LIN {X 0,Y 355.021,Z 361.259,A -85,B 0,C 180,E1 -13509.112,E2 -13509.112} C_VEL
LIN {X 0,Y 354.928,Z 361.272,A -85,B 0,C 180,E1 -13512.581,E2 -13512.581} C_VEL
LIN {X 0,Y 354.896,Z 361.279,A -85,B 0,C 180,E1 -13516.096,E2 -13516.096} C_VEL
LIN {X 0,Y 354.913,Z 361.273,A -85,B 0,C 180,E1 -13518.472,E2 -13518.472} C_VEL
LIN {X 0,Y 354.841,Z 361.284,A -85,B 0,C 180,E1 -13522.106,E2 -13522.106} C_VEL
LIN {X 0,Y 354.905,Z 361.279,A -85,B 0,C 180,E1 -13525.827,E2 -13525.827} C_VEL
LIN {X 0,Y 354.852,Z 361.286,A -85,B 0,C 180,E1 -13529.679,E2 -13529.679} C_VEL
LIN {X 0,Y 354.812,Z 361.29,A -85,B 0,C 180,E1 -13533.702,E2 -13533.702} C_VEL
LIN {X 0,Y 354.806,Z 361.286,A -85,B 0,C 180,E1 -13536.459,E2 -13536.459} C_VEL
LIN {X 0,Y 354.83,Z 361.289,A -85,B 0,C 180,E1 -13539.423,E2 -13539.423} C_VEL
LIN {X 0,Y 354.794,Z 361.289,A -85,B 0,C 180,E1 -13542.867,E2 -13542.867} C_VEL
LIN {X 0,Y 354.786,Z 361.288,A -85,B 0,C 180,E1 -13546.106,E2 -13546.106} C_VEL
LIN {X 0,Y 354.794,Z 361.293,A -85,B 0,C 180,E1 -13549.179,E2 -13549.179} C_VEL
LIN {X 0,Y 354.813,Z 361.285,A -85,B 0,C 180,E1 -13552.402,E2 -13552.402} C_VEL
LIN {X 0,Y 354.818,Z 361.288,A -85,B 0,C 180,E1 -13554.941,E2 -13554.941} C_VEL
LIN {X 0,Y 354.799,Z 361.287,A -85,B 0,C 180,E1 -13558.405,E2 -13558.405} C_VEL
LIN {X 0,Y 354.855,Z 361.281,A -85,B 0,C 180,E1 -13561.618,E2 -13561.618} C_VEL
LIN {X 0,Y 354.905,Z 361.274,A -85,B 0,C 180,E1 -13564.172,E2 -13564.172} C_VEL
LIN {X 0,Y 354.841,Z 361.281,A -85,B 0,C 180,E1 -13567.894,E2 -13567.894} C_VEL
LIN {X 0,Y 354.928,Z 361.271,A -85,B 0,C 180,E1 -13571.891,E2 -13571.891} C_VEL
LIN {X 0,Y 354.949,Z 361.268,A -85,B 0,C 180,E1 -13575.98,E2 -13575.98} C_VEL
LIN {X 0,Y 354.974,Z 361.419,A -85,B 0,C 180,E1 -13578.978,E2 -13578.978} C_VEL
LIN {X 0,Y 358.596,Z 373.086,A -85,B 0,C 180,E1 -13579.84,E2 -13579.84} C_VEL
LIN {X 0,Y 360.664,Z 380.509,A -85,B 0,C 180,E1 -13580.491,E2 -13580.491} C_VEL
LIN {X 0,Y 359.761,Z 392.776,A -85,B 0,C 180,E1 -13581.574,E2 -13581.574} C_VEL
LIN {X 0,Y 358.877,Z 403.838,A -85,B 0,C 180,E1 -13582.827,E2 -13582.827} C_VEL
LIN {X 0,Y 358.135,Z 412.74,A -85,B 0,C 180,E1 -13584.086,E2 -13584.086} C_VEL
LIN {X 0,Y 357.355,Z 420.912,A -85,B 0,C 180,E1 -13585.487,E2 -13585.487} C_VEL
LIN {X 0,Y 356.477,Z 428.926,A -85,B 0,C 180,E1 -13587.174,E2 -13587.174} C_VEL
LIN {X 0,Y 355.809,Z 435.373,A -85,B 0,C 180,E1 -13588.867,E2 -13588.867} C_VEL
LIN {X 0,Y 355.327,Z 440.508,A -85,B 0,C 180,E1 -13590.566,E2 -13590.566} C_VEL
LIN {X 0,Y 354.88,Z 444.523,A -85,B 0,C 180,E1 -13592.269,E2 -13592.269} C_VEL
LIN {X 0,Y 354.623,Z 446.627,A -85,B 0,C 180,E1 -13593.408,E2 -13593.408} C_VEL
LIN {X 0,Y 354.558,Z 449.523,A -85,B 0,C 180,E1 -13595.687,E2 -13595.687} C_VEL
LIN {X 0,Y 354.54,Z 450.755,A -85,B 0,C 180,E1 -13597.626,E2 -13597.626} C_VEL
LIN {X 0,Y 354.539,Z 450.924,A -85,B 0,C 180,E1 -13599.124,E2 -13599.124} C_VEL
LIN {X 0,Y 354.762,Z 449.92,A -85,B 0,C 180,E1 -13601.425,E2 -13601.425} C_VEL
LIN {X 0,Y 354.949,Z 448.782,A -85,B 0,C 180,E1 -13602.579,E2 -13602.579} C_VEL
LIN {X 0,Y 355.473,Z 446.222,A -85,B 0,C 180,E1 -13604.354,E2 -13604.354} C_VEL
LIN {X 0,Y 356.044,Z 442.817,A -85,B 0,C 180,E1 -13606.042,E2 -13606.042} C_VEL
LIN {X 0,Y 356.747,Z 438.198,A -85,B 0,C 180,E1 -13607.779,E2 -13607.779} C_VEL
LIN {X 0,Y 357.852,Z 431.183,A -85,B 0,C 180,E1 -13609.802,E2 -13609.802} C_VEL
LIN {X 0,Y 359.004,Z 423.471,A -85,B 0,C 180,E1 -13611.533,E2 -13611.533} C_VEL
LIN {X 0,Y 360.247,Z 414.193,A -85,B 0,C 180,E1 -13613.19,E2 -13613.19} C_VEL
LIN {X 0,Y 361.309,Z 404.665,A -85,B 0,C 180,E1 -13614.567,E2 -13614.567} C_VEL
LIN {X 0,Y 362.351,Z 394.731,A -85,B 0,C 180,E1 -13615.719,E2 -13615.719} C_VEL
LIN {X 0,Y 363.291,Z 385.09,A -85,B 0,C 180,E1 -13616.62,E2 -13616.62} C_VEL
LIN {X 0,Y 359.553,Z 373.52,A -85,B 0,C 180,E1 -13617.813,E2 -13617.813} C_VEL
LIN {X 0,Y 354.995,Z 361.878,A -85,B 0,C 180,E1 -13618.848,E2 -13618.848} C_VEL
LIN {X 0,Y 354.862,Z 361.284,A -85,B 0,C 180,E1 -13618.947,E2 -13618.947} C_VEL
LIN {X 0,Y 354.788,Z 361.299,A -85,B 0,C 180,E1 -13622.332,E2 -13622.332} C_VEL
LIN {X 0,Y 354.822,Z 361.291,A -85,B 0,C 180,E1 -13625.698,E2 -13625.698} C_VEL
LIN {X 0,Y 354.824,Z 361.288,A -85,B 0,C 180,E1 -13629.423,E2 -13629.423} C_VEL
LIN {X 0,Y 354.779,Z 361.293,A -85,B 0,C 180,E1 -13631.346,E2 -13631.346} C_VEL
LIN {X 0,Y 354.081,Z 361.38,A -85,B 0,C 180,E1 -13632.293,E2 -13632.293} C_VEL
LIN {X 0,Y 351.182,Z 361.741,A -85,B 0,C 180,E1 -13633.831,E2 -13633.831} C_VEL
LIN {X 0,Y 348.77,Z 362.043,A -85,B 0,C 180,E1 -13635.076,E2 -13635.076} C_VEL
LIN {X 0,Y 347.779,Z 362.167,A -85,B 0,C 180,E1 -13636.04,E2 -13636.04} C_VEL
LIN {X 0,Y 347.721,Z 362.17,A -85,B 0,C 180,E1 -13636.367,E2 -13636.367} C_VEL
LIN {X 0,Y 347.754,Z 362.168,A -85,B 0,C 180,E1 -13639.705,E2 -13639.705} C_VEL
LIN {X 0,Y 347.765,Z 362.167,A -85,B 0,C 180,E1 -13642.679,E2 -13642.679} C_VEL
LIN {X 0,Y 347.746,Z 362.17,A -85,B 0,C 180,E1 -13645.955,E2 -13645.955} C_VEL
LIN {X 0,Y 347.768,Z 362.134,A -85,B 0,C 180,E1 -13649.653,E2 -13649.653} C_VEL
LIN {X 0,Y 347.85,Z 362.149,A -85,B 0,C 180,E1 -13652.744,E2 -13652.744} C_VEL
LIN {X 0,Y 347.785,Z 362.157,A -85,B 0,C 180,E1 -13656.161,E2 -13656.161} C_VEL
LIN {X 0,Y 347.814,Z 362.16,A -85,B 0,C 180,E1 -13659.909,E2 -13659.909} C_VEL
LIN {X 0,Y 347.863,Z 362.145,A -85,B 0,C 180,E1 -13662.359,E2 -13662.359} C_VEL
LIN {X 0,Y 347.894,Z 362.151,A -85,B 0,C 180,E1 -13665.97,E2 -13665.97} C_VEL
LIN {X 0,Y 347.93,Z 362.144,A -85,B 0,C 180,E1 -13669.525,E2 -13669.525} C_VEL
LIN {X 0,Y 348.071,Z 362.129,A -85,B 0,C 180,E1 -13671.874,E2 -13671.874} C_VEL
LIN {X 0,Y 348.065,Z 362.118,A -85,B 0,C 180,E1 -13674.205,E2 -13674.205} C_VEL
LIN {X 0,Y 348.205,Z 362.112,A -85,B 0,C 180,E1 -13677.686,E2 -13677.686} C_VEL
LIN {X 0,Y 348.365,Z 362.082,A -85,B 0,C 180,E1 -13680,E2 -13680} C_VEL
LIN {X 0,Y 348.205,Z 362.113,A -85,B 0,C 180,E1 -13682.313,E2 -13682.313} C_VEL
LIN {X 0,Y 348.102,Z 362.124,A -85,B 0,C 180,E1 -13686.957,E2 -13686.957} C_VEL
LIN {X 0,Y 347.963,Z 362.136,A -85,B 0,C 180,E1 -13689.298,E2 -13689.298} C_VEL
LIN {X 0,Y 347.886,Z 362.15,A -85,B 0,C 180,E1 -13692.839,E2 -13692.839} C_VEL
LIN {X 0,Y 347.835,Z 362.158,A -85,B 0,C 180,E1 -13696.431,E2 -13696.431} C_VEL
LIN {X 0,Y 347.851,Z 362.156,A -85,B 0,C 180,E1 -13698.86,E2 -13698.86} C_VEL
LIN {X 0,Y 347.77,Z 362.168,A -85,B 0,C 180,E1 -13702.579,E2 -13702.579} C_VEL
LIN {X 0,Y 347.808,Z 362.165,A -85,B 0,C 180,E1 -13705.109,E2 -13705.109} C_VEL
LIN {X 0,Y 347.808,Z 362.165,A -85,B 0,C 180,E1 -13707.694,E2 -13707.694} C_VEL
LIN {X 0,Y 347.76,Z 362.171,A -85,B 0,C 180,E1 -13710.347,E2 -13710.347} C_VEL
LIN {X 0,Y 347.741,Z 362.171,A -85,B 0,C 180,E1 -13714.464,E2 -13714.464} C_VEL
LIN {X 0,Y 347.776,Z 362.156,A -85,B 0,C 180,E1 -13717.99,E2 -13717.99} C_VEL
LIN {X 0,Y 347.78,Z 362.155,A -85,B 0,C 180,E1 -13721.826,E2 -13721.826} C_VEL
LIN {X 0,Y 347.797,Z 362.164,A -85,B 0,C 180,E1 -13722.213,E2 -13722.213} C_VEL
LIN {X 0,Y 349.191,Z 369.057,A -85,B 0,C 180,E1 -13725.701,E2 -13725.701} C_VEL
LIN {X 0,Y 350.381,Z 375.055,A -85,B 0,C 180,E1 -13728.555,E2 -13728.555} C_VEL
LIN {X 0,Y 351.655,Z 382.173,A -85,B 0,C 180,E1 -13731.718,E2 -13731.718} C_VEL
LIN {X 0,Y 351.741,Z 385.397,A -85,B 0,C 180,E1 -13733.056,E2 -13733.056} C_VEL
LIN {X 0,Y 350.275,Z 396.112,A -85,B 0,C 180,E1 -13737.199,E2 -13737.199} C_VEL
LIN {X 0,Y 349.041,Z 406.501,A -85,B 0,C 180,E1 -13741.104,E2 -13741.104} C_VEL
LIN {X 0,Y 348.092,Z 416.889,A -85,B 0,C 180,E1 -13744.914,E2 -13744.914} C_VEL
LIN {X 0,Y 347.423,Z 425.713,A -85,B 0,C 180,E1 -13748.105,E2 -13748.105} C_VEL
LIN {X 0,Y 350.097,Z 440.51,A -85,B 0,C 180,E1 -13748.818,E2 -13748.818} C_VEL
LIN {X 0,Y 351.654,Z 453.114,A -85,B 0,C 180,E1 -13749.614,E2 -13749.614} C_VEL
LIN {X 0,Y 352.322,Z 464.451,A -85,B 0,C 180,E1 -13750.489,E2 -13750.489} C_VEL
LIN {X 0,Y 352.267,Z 477.128,A -85,B 0,C 180,E1 -13751.687,E2 -13751.687} C_VEL
LIN {X 0,Y 351.127,Z 487.251,A -85,B 0,C 180,E1 -13752.83,E2 -13752.83} C_VEL
LIN {X 0,Y 349.685,Z 497.503,A -85,B 0,C 180,E1 -13754.258,E2 -13754.258} C_VEL
LIN {X 0,Y 348.829,Z 505.758,A -85,B 0,C 180,E1 -13755.677,E2 -13755.677} C_VEL
LIN {X 0,Y 347.695,Z 514.218,A -85,B 0,C 180,E1 -13757.451,E2 -13757.451} C_VEL
LIN {X 0,Y 346.983,Z 520.939,A -85,B 0,C 180,E1 -13759.202,E2 -13759.202} C_VEL
LIN {X 0,Y 346.652,Z 527.13,A -85,B 0,C 180,E1 -13761.255,E2 -13761.255} C_VEL
LIN {X 0,Y 346.637,Z 532.039,A -85,B 0,C 180,E1 -13763.447,E2 -13763.447} C_VEL
LIN {X 0,Y 346.765,Z 535.029,A -85,B 0,C 180,E1 -13765.351,E2 -13765.351} C_VEL
LIN {X 0,Y 346.931,Z 536.325,A -85,B 0,C 180,E1 -13766.517,E2 -13766.517} C_VEL
LIN {X 0,Y 346.964,Z 537.152,A -85,B 0,C 180,E1 -13767.679,E2 -13767.679} C_VEL
LIN {X 0,Y 347.059,Z 537.594,A -85,B 0,C 180,E1 -13770.001,E2 -13770.001} C_VEL
LIN {X 0,Y 347.019,Z 537.206,A -85,B 0,C 180,E1 -13771.161,E2 -13771.161} C_VEL
LIN {X 0,Y 347.012,Z 536.375,A -85,B 0,C 180,E1 -13772.322,E2 -13772.322} C_VEL
LIN {X 0,Y 347.078,Z 535.124,A -85,B 0,C 180,E1 -13773.484,E2 -13773.484} C_VEL
LIN {X 0,Y 346.836,Z 532.39,A -85,B 0,C 180,E1 -13775.233,E2 -13775.233} C_VEL
LIN {X 0,Y 346.749,Z 528.611,A -85,B 0,C 180,E1 -13776.986,E2 -13776.986} C_VEL
LIN {X 0,Y 346.752,Z 523.674,A -85,B 0,C 180,E1 -13778.744,E2 -13778.744} C_VEL
LIN {X 0,Y 346.95,Z 517.446,A -85,B 0,C 180,E1 -13780.505,E2 -13780.505} C_VEL
LIN {X 0,Y 347.514,Z 509.73,A -85,B 0,C 180,E1 -13782.261,E2 -13782.261} C_VEL
LIN {X 0,Y 348.231,Z 501.871,A -85,B 0,C 180,E1 -13783.719,E2 -13783.719} C_VEL
LIN {X 0,Y 348.864,Z 494.15,A -85,B 0,C 180,E1 -13784.913,E2 -13784.913} C_VEL
LIN {X 0,Y 349.834,Z 484.267,A -85,B 0,C 180,E1 -13786.186,E2 -13786.186} C_VEL
LIN {X 0,Y 350.586,Z 474.636,A -85,B 0,C 180,E1 -13787.199,E2 -13787.199} C_VEL
LIN {X 0,Y 350.156,Z 462.196,A -85,B 0,C 180,E1 -13788.278,E2 -13788.278} C_VEL
LIN {X 0,Y 349.338,Z 449.493,A -85,B 0,C 180,E1 -13789.136,E2 -13789.136} C_VEL
LIN {X 0,Y 348.224,Z 436.683,A -85,B 0,C 180,E1 -13789.778,E2 -13789.778} C_VEL
LIN {X 0,Y 347.061,Z 426.898,A -85,B 0,C 180,E1 -13790.137,E2 -13790.137} C_VEL
LIN {X 0,Y 347.661,Z 415.33,A -85,B 0,C 180,E1 -13794.205,E2 -13794.205} C_VEL
LIN {X 0,Y 348.503,Z 403.834,A -85,B 0,C 180,E1 -13798.289,E2 -13798.289} C_VEL
LIN {X 0,Y 349.388,Z 393.64,A -85,B 0,C 180,E1 -13801.955,E2 -13801.955} C_VEL
LIN {X 0,Y 350.621,Z 382.261,A -85,B 0,C 180,E1 -13806.148,E2 -13806.148} C_VEL
LIN {X 0,Y 350.742,Z 378.306,A -85,B 0,C 180,E1 -13807.673,E2 -13807.673} C_VEL
LIN {X 0,Y 349.416,Z 370.597,A -85,B 0,C 180,E1 -13810.852,E2 -13810.852} C_VEL
LIN {X 0,Y 347.922,Z 362.984,A -85,B 0,C 180,E1 -13814.185,E2 -13814.185} C_VEL
LIN {X 0,Y 347.794,Z 362.167,A -85,B 0,C 180,E1 -13814.577,E2 -13814.577} C_VEL
LIN {X 0,Y 347.754,Z 362.165,A -85,B 0,C 180,E1 -13818.398,E2 -13818.398} C_VEL
LIN {X 0,Y 347.778,Z 362.161,A -85,B 0,C 180,E1 -13822.012,E2 -13822.012} C_VEL
LIN {X 0,Y 347.749,Z 362.165,A -85,B 0,C 180,E1 -13825.537,E2 -13825.537} C_VEL
LIN {X 0,Y 347.749,Z 362.166,A -85,B 0,C 180,E1 -13828.301,E2 -13828.301} C_VEL
LIN {X 0,Y 347.783,Z 362.164,A -85,B 0,C 180,E1 -13830.988,E2 -13830.988} C_VEL
LIN {X 0,Y 347.836,Z 362.154,A -85,B 0,C 180,E1 -13833.608,E2 -13833.608} C_VEL
LIN {X 0,Y 347.794,Z 362.16,A -85,B 0,C 180,E1 -13836.162,E2 -13836.162} C_VEL
LIN {X 0,Y 347.818,Z 362.157,A -85,B 0,C 180,E1 -13839.91,E2 -13839.91} C_VEL
LIN {X 0,Y 347.871,Z 362.153,A -85,B 0,C 180,E1 -13842.36,E2 -13842.36} C_VEL
LIN {X 0,Y 347.903,Z 362.147,A -85,B 0,C 180,E1 -13845.971,E2 -13845.971} C_VEL
LIN {X 0,Y 347.934,Z 362.142,A -85,B 0,C 180,E1 -13849.526,E2 -13849.526} C_VEL
LIN {X 0,Y 348.114,Z 362.12,A -85,B 0,C 180,E1 -13853.043,E2 -13853.043} C_VEL
LIN {X 0,Y 348.211,Z 362.108,A -85,B 0,C 180,E1 -13857.687,E2 -13857.687} C_VEL
LIN {X 0,Y 348.352,Z 362.093,A -85,B 0,C 180,E1 -13860,E2 -13860} C_VEL
LIN {X 0,Y 348.212,Z 362.112,A -85,B 0,C 180,E1 -13862.314,E2 -13862.314} C_VEL
LIN {X 0,Y 348.112,Z 362.119,A -85,B 0,C 180,E1 -13866.958,E2 -13866.958} C_VEL
LIN {X 0,Y 347.974,Z 362.137,A -85,B 0,C 180,E1 -13869.299,E2 -13869.299} C_VEL
LIN {X 0,Y 347.896,Z 362.146,A -85,B 0,C 180,E1 -13872.84,E2 -13872.84} C_VEL
LIN {X 0,Y 347.845,Z 362.154,A -85,B 0,C 180,E1 -13876.431,E2 -13876.431} C_VEL
LIN {X 0,Y 347.862,Z 362.15,A -85,B 0,C 180,E1 -13878.86,E2 -13878.86} C_VEL
LIN {X 0,Y 347.78,Z 362.161,A -85,B 0,C 180,E1 -13882.579,E2 -13882.579} C_VEL
LIN {X 0,Y 347.818,Z 362.157,A -85,B 0,C 180,E1 -13885.108,E2 -13885.108} C_VEL
LIN {X 0,Y 347.814,Z 362.163,A -85,B 0,C 180,E1 -13887.694,E2 -13887.694} C_VEL
LIN {X 0,Y 347.767,Z 362.163,A -85,B 0,C 180,E1 -13890.347,E2 -13890.347} C_VEL
LIN {X 0,Y 347.75,Z 362.164,A -85,B 0,C 180,E1 -13894.464,E2 -13894.464} C_VEL
LIN {X 0,Y 347.782,Z 362.162,A -85,B 0,C 180,E1 -13897.989,E2 -13897.989} C_VEL
LIN {X 0,Y 347.757,Z 362.166,A -85,B 0,C 180,E1 -13901.83,E2 -13901.83} C_VEL
LIN {X 0,Y 347.772,Z 362.165,A -85,B 0,C 180,E1 -13905.017,E2 -13905.017} C_VEL
LIN {X 0,Y 347.756,Z 362.164,A -85,B 0,C 180,E1 -13908.397,E2 -13908.397} C_VEL
LIN {X 0,Y 347.78,Z 362.161,A -85,B 0,C 180,E1 -13912.011,E2 -13912.011} C_VEL
LIN {X 0,Y 347.75,Z 362.167,A -85,B 0,C 180,E1 -13915.536,E2 -13915.536} C_VEL
LIN {X 0,Y 347.77,Z 362.163,A -85,B 0,C 180,E1 -13919.653,E2 -13919.653} C_VEL
LIN {X 0,Y 347.857,Z 362.155,A -85,B 0,C 180,E1 -13922.744,E2 -13922.744} C_VEL
LIN {X 0,Y 347.795,Z 362.159,A -85,B 0,C 180,E1 -13926.161,E2 -13926.161} C_VEL
LIN {X 0,Y 347.819,Z 362.156,A -85,B 0,C 180,E1 -13929.909,E2 -13929.909} C_VEL
LIN {X 0,Y 347.872,Z 362.151,A -85,B 0,C 180,E1 -13932.359,E2 -13932.359} C_VEL
LIN {X 0,Y 347.903,Z 362.146,A -85,B 0,C 180,E1 -13935.97,E2 -13935.97} C_VEL
LIN {X 0,Y 347.931,Z 362.337,A -85,B 0,C 180,E1 -13938.64,E2 -13938.64} C_VEL
LIN {X 0,Y 351.521,Z 373.703,A -85,B 0,C 180,E1 -13939.502,E2 -13939.502} C_VEL
LIN {X 0,Y 353.811,Z 381.971,A -85,B 0,C 180,E1 -13940.247,E2 -13940.247} C_VEL
LIN {X 0,Y 352.949,Z 393.281,A -85,B 0,C 180,E1 -13941.266,E2 -13941.266} C_VEL
LIN {X 0,Y 352.034,Z 404.422,A -85,B 0,C 180,E1 -13942.543,E2 -13942.543} C_VEL
LIN {X 0,Y 351.159,Z 414.255,A -85,B 0,C 180,E1 -13943.968,E2 -13943.968} C_VEL
LIN {X 0,Y 350.215,Z 423.775,A -85,B 0,C 180,E1 -13945.683,E2 -13945.683} C_VEL
LIN {X 0,Y 349.335,Z 431.411,A -85,B 0,C 180,E1 -13947.405,E2 -13947.405} C_VEL
LIN {X 0,Y 348.585,Z 438.404,A -85,B 0,C 180,E1 -13949.422,E2 -13949.422} C_VEL
LIN {X 0,Y 348.098,Z 443.08,A -85,B 0,C 180,E1 -13951.156,E2 -13951.156} C_VEL
LIN {X 0,Y 347.72,Z 446.676,A -85,B 0,C 180,E1 -13952.895,E2 -13952.895} C_VEL
LIN {X 0,Y 347.543,Z 449.272,A -85,B 0,C 180,E1 -13954.639,E2 -13954.639} C_VEL
LIN {X 0,Y 347.516,Z 450.499,A -85,B 0,C 180,E1 -13955.803,E2 -13955.803} C_VEL
LIN {X 0,Y 347.49,Z 451.631,A -85,B 0,C 180,E1 -13957.677,E2 -13957.677} C_VEL
LIN {X 0,Y 347.527,Z 451.784,A -85,B 0,C 180,E1 -13959.31,E2 -13959.31} C_VEL
LIN {X 0,Y 347.61,Z 451.448,A -85,B 0,C 180,E1 -13960.483,E2 -13960.483} C_VEL
LIN {X 0,Y 347.763,Z 450.703,A -85,B 0,C 180,E1 -13961.658,E2 -13961.658} C_VEL
LIN {X 0,Y 347.981,Z 449.527,A -85,B 0,C 180,E1 -13962.835,E2 -13962.835} C_VEL
LIN {X 0,Y 348.492,Z 447.114,A -85,B 0,C 180,E1 -13964.529,E2 -13964.529} C_VEL
LIN {X 0,Y 349.148,Z 443.435,A -85,B 0,C 180,E1 -13966.367,E2 -13966.367} C_VEL
LIN {X 0,Y 349.912,Z 438.745,A -85,B 0,C 180,E1 -13968.138,E2 -13968.138} C_VEL
LIN {X 0,Y 350.913,Z 432.759,A -85,B 0,C 180,E1 -13969.905,E2 -13969.905} C_VEL
LIN {X 0,Y 352.103,Z 425.256,A -85,B 0,C 180,E1 -13971.669,E2 -13971.669} C_VEL
LIN {X 0,Y 353.213,Z 417.516,A -85,B 0,C 180,E1 -13973.139,E2 -13973.139} C_VEL
LIN {X 0,Y 354.387,Z 407.977,A -85,B 0,C 180,E1 -13974.61,E2 -13974.61} C_VEL
LIN {X 0,Y 355.626,Z 397.404,A -85,B 0,C 180,E1 -13975.915,E2 -13975.915} C_VEL
LIN {X 0,Y 356.659,Z 386.918,A -85,B 0,C 180,E1 -13976.949,E2 -13976.949} C_VEL
LIN {X 0,Y 353.253,Z 376.293,A -85,B 0,C 180,E1 -13978.104,E2 -13978.104} C_VEL
LIN {X 0,Y 348.435,Z 364.327,A -85,B 0,C 180,E1 -13979.24,E2 -13979.24} C_VEL
LIN {X 0,Y 347.781,Z 362.17,A -85,B 0,C 180,E1 -13979.446,E2 -13979.446} C_VEL
LIN {X 0,Y 347.733,Z 362.172,A -85,B 0,C 180,E1 -13983.071,E2 -13983.071} C_VEL
LIN {X 0,Y 347.77,Z 362.168,A -85,B 0,C 180,E1 -13986.064,E2 -13986.064} C_VEL
LIN {X 0,Y 347.752,Z 362.171,A -85,B 0,C 180,E1 -13988.792,E2 -13988.792} C_VEL
LIN {X 0,Y 347.75,Z 362.167,A -85,B 0,C 180,E1 -13991.829,E2 -13991.829} C_VEL
LIN {X 0,Y 347.708,Z 362.175,A -85,B 0,C 180,E1 -13995.025,E2 -13995.025} C_VEL
LIN {X 0,Y 347.721,Z 362.17,A -85,B 0,C 180,E1 -13996.367,E2 -13996.367} C_VEL
LIN {X 0,Y 347.104,Z 362.251,A -85,B 0,C 180,E1 -13997.334,E2 -13997.334} C_VEL
LIN {X 0,Y 344.233,Z 362.61,A -85,B 0,C 180,E1 -13998.907,E2 -13998.907} C_VEL
LIN {X 0,Y 341.79,Z 362.909,A -85,B 0,C 180,E1 -14000.181,E2 -14000.181} C_VEL
LIN {X 0,Y 340.774,Z 363.039,A -85,B 0,C 180,E1 -14001.168,E2 -14001.168} C_VEL
LIN {X 0,Y 340.71,Z 363.048,A -85,B 0,C 180,E1 -14001.502,E2 -14001.502} C_VEL
LIN {X 0,Y 340.717,Z 363.045,A -85,B 0,C 180,E1 -14004.72,E2 -14004.72} C_VEL
LIN {X 0,Y 340.714,Z 363.017,A -85,B 0,C 180,E1 -14008.956,E2 -14008.956} C_VEL
LIN {X 0,Y 340.777,Z 363.028,A -85,B 0,C 180,E1 -14012.473,E2 -14012.473} C_VEL
LIN {X 0,Y 340.753,Z 363.036,A -85,B 0,C 180,E1 -14015.638,E2 -14015.638} C_VEL
LIN {X 0,Y 340.753,Z 363.041,A -85,B 0,C 180,E1 -14019.474,E2 -14019.474} C_VEL
LIN {X 0,Y 340.855,Z 363.018,A -85,B 0,C 180,E1 -14021.984,E2 -14021.984} C_VEL
LIN {X 0,Y 340.865,Z 363.026,A -85,B 0,C 180,E1 -14025.704,E2 -14025.704} C_VEL
LIN {X 0,Y 340.872,Z 363.024,A -85,B 0,C 180,E1 -14029.306,E2 -14029.306} C_VEL
LIN {X 0,Y 341.072,Z 362.997,A -85,B 0,C 180,E1 -14032.898,E2 -14032.898} C_VEL
LIN {X 0,Y 341.167,Z 362.988,A -85,B 0,C 180,E1 -14037.638,E2 -14037.638} C_VEL
LIN {X 0,Y 341.314,Z 362.96,A -85,B 0,C 180,E1 -14040,E2 -14040} C_VEL
LIN {X 0,Y 341.167,Z 362.99,A -85,B 0,C 180,E1 -14042.361,E2 -14042.361} C_VEL
LIN {X 0,Y 341.072,Z 363.001,A -85,B 0,C 180,E1 -14047.102,E2 -14047.102} C_VEL
LIN {X 0,Y 340.867,Z 363.022,A -85,B 0,C 180,E1 -14050.694,E2 -14050.694} C_VEL
LIN {X 0,Y 340.858,Z 363.021,A -85,B 0,C 180,E1 -14054.325,E2 -14054.325} C_VEL
LIN {X 0,Y 340.833,Z 363.029,A -85,B 0,C 180,E1 -14058.467,E2 -14058.467} C_VEL
LIN {X 0,Y 340.749,Z 363.042,A -85,B 0,C 180,E1 -14061.857,E2 -14061.857} C_VEL
LIN {X 0,Y 340.769,Z 363.041,A -85,B 0,C 180,E1 -14065.665,E2 -14065.665} C_VEL
LIN {X 0,Y 340.738,Z 363.045,A -85,B 0,C 180,E1 -14068.32,E2 -14068.32} C_VEL
LIN {X 0,Y 340.7,Z 363.049,A -85,B 0,C 180,E1 -14071.044,E2 -14071.044} C_VEL
LIN {X 0,Y 340.715,Z 363.044,A -85,B 0,C 180,E1 -14075.279,E2 -14075.279} C_VEL
LIN {X 0,Y 340.716,Z 363.033,A -85,B 0,C 180,E1 -14078.389,E2 -14078.389} C_VEL
LIN {X 0,Y 340.764,Z 363.119,A -85,B 0,C 180,E1 -14081.701,E2 -14081.701} C_VEL
LIN {X 0,Y 342.074,Z 369.494,A -85,B 0,C 180,E1 -14085.041,E2 -14085.041} C_VEL
LIN {X 0,Y 343.401,Z 376.226,A -85,B 0,C 180,E1 -14088.319,E2 -14088.319} C_VEL
LIN {X 0,Y 344.686,Z 383.399,A -85,B 0,C 180,E1 -14091.588,E2 -14091.588} C_VEL
LIN {X 0,Y 344.839,Z 385.866,A -85,B 0,C 180,E1 -14092.64,E2 -14092.64} C_VEL
LIN {X 0,Y 343.457,Z 395.449,A -85,B 0,C 180,E1 -14096.463,E2 -14096.463} C_VEL
LIN {X 0,Y 342.136,Z 405.829,A -85,B 0,C 180,E1 -14100.463,E2 -14100.463} C_VEL
LIN {X 0,Y 341.152,Z 416.18,A -85,B 0,C 180,E1 -14104.367,E2 -14104.367} C_VEL
LIN {X 0,Y 340.455,Z 424.893,A -85,B 0,C 180,E1 -14107.57,E2 -14107.57} C_VEL
LIN {X 0,Y 343.155,Z 439.246,A -85,B 0,C 180,E1 -14108.286,E2 -14108.286} C_VEL
LIN {X 0,Y 344.743,Z 451.758,A -85,B 0,C 180,E1 -14109.091,E2 -14109.091} C_VEL
LIN {X 0,Y 345.479,Z 463.306,A -85,B 0,C 180,E1 -14110.003,E2 -14110.003} C_VEL
LIN {X 0,Y 345.44,Z 475.363,A -85,B 0,C 180,E1 -14111.158,E2 -14111.158} C_VEL
LIN {X 0,Y 344.857,Z 483.284,A -85,B 0,C 180,E1 -14112.048,E2 -14112.048} C_VEL
LIN {X 0,Y 343.333,Z 493.137,A -85,B 0,C 180,E1 -14113.348,E2 -14113.348} C_VEL
LIN {X 0,Y 342.02,Z 503.004,A -85,B 0,C 180,E1 -14114.968,E2 -14114.968} C_VEL
LIN {X 0,Y 341.233,Z 509.666,A -85,B 0,C 180,E1 -14116.3,E2 -14116.3} C_VEL
LIN {X 0,Y 340.326,Z 517.087,A -85,B 0,C 180,E1 -14118.083,E2 -14118.083} C_VEL
LIN {X 0,Y 339.753,Z 523.084,A -85,B 0,C 180,E1 -14119.874,E2 -14119.874} C_VEL
LIN {X 0,Y 339.543,Z 527.863,A -85,B 0,C 180,E1 -14121.67,E2 -14121.67} C_VEL
LIN {X 0,Y 339.561,Z 531.518,A -85,B 0,C 180,E1 -14123.449,E2 -14123.449} C_VEL
LIN {X 0,Y 339.682,Z 534.216,A -85,B 0,C 180,E1 -14125.254,E2 -14125.254} C_VEL
LIN {X 0,Y 339.857,Z 535.491,A -85,B 0,C 180,E1 -14126.444,E2 -14126.444} C_VEL
LIN {X 0,Y 339.915,Z 536.3,A -85,B 0,C 180,E1 -14127.631,E2 -14127.631} C_VEL
LIN {X 0,Y 340.013,Z 536.714,A -85,B 0,C 180,E1 -14130.001,E2 -14130.001} C_VEL
LIN {X 0,Y 339.971,Z 536.306,A -85,B 0,C 180,E1 -14131.185,E2 -14131.185} C_VEL
LIN {X 0,Y 339.966,Z 535.449,A -85,B 0,C 180,E1 -14132.37,E2 -14132.37} C_VEL
LIN {X 0,Y 340.033,Z 534.182,A -85,B 0,C 180,E1 -14133.556,E2 -14133.556} C_VEL
LIN {X 0,Y 339.761,Z 531.411,A -85,B 0,C 180,E1 -14135.342,E2 -14135.342} C_VEL
LIN {X 0,Y 339.693,Z 527.597,A -85,B 0,C 180,E1 -14137.132,E2 -14137.132} C_VEL
LIN {X 0,Y 339.684,Z 522.618,A -85,B 0,C 180,E1 -14138.928,E2 -14138.928} C_VEL
LIN {X 0,Y 339.917,Z 516.348,A -85,B 0,C 180,E1 -14140.725,E2 -14140.725} C_VEL
LIN {X 0,Y 340.506,Z 508.583,A -85,B 0,C 180,E1 -14142.517,E2 -14142.517} C_VEL
LIN {X 0,Y 341.22,Z 500.655,A -85,B 0,C 180,E1 -14144.006,E2 -14144.006} C_VEL
LIN {X 0,Y 342.196,Z 490.991,A -85,B 0,C 180,E1 -14145.486,E2 -14145.486} C_VEL
LIN {X 0,Y 343.195,Z 480.271,A -85,B 0,C 180,E1 -14146.814,E2 -14146.814} C_VEL
LIN {X 0,Y 343.567,Z 474.633,A -85,B 0,C 180,E1 -14147.409,E2 -14147.409} C_VEL
LIN {X 0,Y 343.206,Z 462.733,A -85,B 0,C 180,E1 -14148.492,E2 -14148.492} C_VEL
LIN {X 0,Y 342.438,Z 450.27,A -85,B 0,C 180,E1 -14149.377,E2 -14149.377} C_VEL
LIN {X 0,Y 341.333,Z 437.111,A -85,B 0,C 180,E1 -14150.077,E2 -14150.077} C_VEL
LIN {X 0,Y 339.999,Z 426.09,A -85,B 0,C 180,E1 -14150.495,E2 -14150.495} C_VEL
LIN {X 0,Y 340.666,Z 414.112,A -85,B 0,C 180,E1 -14154.807,E2 -14154.807} C_VEL
LIN {X 0,Y 341.552,Z 402.834,A -85,B 0,C 180,E1 -14158.919,E2 -14158.919} C_VEL
LIN {X 0,Y 342.41,Z 393.793,A -85,B 0,C 180,E1 -14162.254,E2 -14162.254} C_VEL
LIN {X 0,Y 343.649,Z 382.869,A -85,B 0,C 180,E1 -14166.377,E2 -14166.377} C_VEL
LIN {X 0,Y 343.707,Z 379.2,A -85,B 0,C 180,E1 -14167.839,E2 -14167.839} C_VEL
LIN {X 0,Y 342.386,Z 371.552,A -85,B 0,C 180,E1 -14171.061,E2 -14171.061} C_VEL
LIN {X 0,Y 340.857,Z 363.569,A -85,B 0,C 180,E1 -14174.648,E2 -14174.648} C_VEL
LIN {X 0,Y 340.746,Z 363.043,A -85,B 0,C 180,E1 -14174.983,E2 -14174.983} C_VEL
LIN {X 0,Y 340.69,Z 363.047,A -85,B 0,C 180,E1 -14178.691,E2 -14178.691} C_VEL
LIN {X 0,Y 340.737,Z 363.038,A -85,B 0,C 180,E1 -14181.773,E2 -14181.773} C_VEL
LIN {X 0,Y 340.727,Z 363.04,A -85,B 0,C 180,E1 -14185.596,E2 -14185.596} C_VEL
LIN {X 0,Y 340.702,Z 363.047,A -85,B 0,C 180,E1 -14188.956,E2 -14188.956} C_VEL
LIN {X 0,Y 340.808,Z 363.033,A -85,B 0,C 180,E1 -14193.02,E2 -14193.02} C_VEL
LIN {X 0,Y 340.761,Z 363.035,A -85,B 0,C 180,E1 -14195.639,E2 -14195.639} C_VEL
LIN {X 0,Y 340.758,Z 363.036,A -85,B 0,C 180,E1 -14199.475,E2 -14199.475} C_VEL
LIN {X 0,Y 340.863,Z 363.024,A -85,B 0,C 180,E1 -14201.985,E2 -14201.985} C_VEL
LIN {X 0,Y 340.875,Z 363.021,A -85,B 0,C 180,E1 -14205.705,E2 -14205.705} C_VEL
LIN {X 0,Y 340.876,Z 363.021,A -85,B 0,C 180,E1 -14209.307,E2 -14209.307} C_VEL
LIN {X 0,Y 341.083,Z 362.996,A -85,B 0,C 180,E1 -14212.899,E2 -14212.899} C_VEL
LIN {X 0,Y 341.173,Z 362.984,A -85,B 0,C 180,E1 -14217.639,E2 -14217.639} C_VEL
LIN {X 0,Y 341.303,Z 362.971,A -85,B 0,C 180,E1 -14220,E2 -14220} C_VEL
LIN {X 0,Y 341.173,Z 362.988,A -85,B 0,C 180,E1 -14222.361,E2 -14222.361} C_VEL
LIN {X 0,Y 341.082,Z 362.995,A -85,B 0,C 180,E1 -14227.102,E2 -14227.102} C_VEL
LIN {X 0,Y 340.877,Z 363.021,A -85,B 0,C 180,E1 -14230.694,E2 -14230.694} C_VEL
LIN {X 0,Y 340.869,Z 363.024,A -85,B 0,C 180,E1 -14234.325,E2 -14234.325} C_VEL
LIN {X 0,Y 340.844,Z 363.026,A -85,B 0,C 180,E1 -14238.467,E2 -14238.467} C_VEL
LIN {X 0,Y 340.76,Z 363.04,A -85,B 0,C 180,E1 -14241.857,E2 -14241.857} C_VEL
LIN {X 0,Y 340.778,Z 363.038,A -85,B 0,C 180,E1 -14245.664,E2 -14245.664} C_VEL
LIN {X 0,Y 340.734,Z 363.039,A -85,B 0,C 180,E1 -14248.321,E2 -14248.321} C_VEL
LIN {X 0,Y 340.709,Z 363.042,A -85,B 0,C 180,E1 -14251.044,E2 -14251.044} C_VEL
LIN {X 0,Y 340.724,Z 363.043,A -85,B 0,C 180,E1 -14255.279,E2 -14255.279} C_VEL
LIN {X 0,Y 340.718,Z 363.04,A -85,B 0,C 180,E1 -14258.386,E2 -14258.386} C_VEL
LIN {X 0,Y 340.705,Z 363.043,A -85,B 0,C 180,E1 -14262.045,E2 -14262.045} C_VEL
LIN {X 0,Y 340.69,Z 363.049,A -85,B 0,C 180,E1 -14265.461,E2 -14265.461} C_VEL
LIN {X 0,Y 340.692,Z 363.045,A -85,B 0,C 180,E1 -14268.69,E2 -14268.69} C_VEL
LIN {X 0,Y 340.739,Z 363.039,A -85,B 0,C 180,E1 -14271.772,E2 -14271.772} C_VEL
LIN {X 0,Y 340.729,Z 363.041,A -85,B 0,C 180,E1 -14275.595,E2 -14275.595} C_VEL
LIN {X 0,Y 340.71,Z 363.046,A -85,B 0,C 180,E1 -14278.956,E2 -14278.956} C_VEL
LIN {X 0,Y 340.784,Z 363.034,A -85,B 0,C 180,E1 -14282.474,E2 -14282.474} C_VEL
LIN {X 0,Y 340.762,Z 363.035,A -85,B 0,C 180,E1 -14285.638,E2 -14285.638} C_VEL
LIN {X 0,Y 340.759,Z 363.036,A -85,B 0,C 180,E1 -14289.474,E2 -14289.474} C_VEL
LIN {X 0,Y 340.863,Z 363.023,A -85,B 0,C 180,E1 -14291.984,E2 -14291.984} C_VEL
LIN {X 0,Y 340.875,Z 363.021,A -85,B 0,C 180,E1 -14295.704,E2 -14295.704} C_VEL
LIN {X 0,Y 340.853,Z 363.026,A -85,B 0,C 180,E1 -14298.266,E2 -14298.266} C_VEL
LIN {X 0,Y 344.947,Z 376.091,A -85,B 0,C 180,E1 -14299.299,E2 -14299.299} C_VEL
LIN {X 0,Y 346.985,Z 383.436,A -85,B 0,C 180,E1 -14299.997,E2 -14299.997} C_VEL
LIN {X 0,Y 346.021,Z 395.178,A -85,B 0,C 180,E1 -14301.09,E2 -14301.09} C_VEL
LIN {X 0,Y 345.097,Z 406.069,A -85,B 0,C 180,E1 -14302.392,E2 -14302.392} C_VEL
LIN {X 0,Y 344.183,Z 415.765,A -85,B 0,C 180,E1 -14303.845,E2 -14303.845} C_VEL
LIN {X 0,Y 343.219,Z 425.174,A -85,B 0,C 180,E1 -14305.595,E2 -14305.595} C_VEL
LIN {X 0,Y 342.317,Z 432.682,A -85,B 0,C 180,E1 -14307.351,E2 -14307.351} C_VEL
LIN {X 0,Y 341.555,Z 439.6,A -85,B 0,C 180,E1 -14309.41,E2 -14309.41} C_VEL
LIN {X 0,Y 341.061,Z 444.207,A -85,B 0,C 180,E1 -14311.18,E2 -14311.18} C_VEL
LIN {X 0,Y 340.647,Z 447.744,A -85,B 0,C 180,E1 -14312.956,E2 -14312.956} C_VEL
LIN {X 0,Y 340.507,Z 450.274,A -85,B 0,C 180,E1 -14314.735,E2 -14314.735} C_VEL
LIN {X 0,Y 340.476,Z 451.472,A -85,B 0,C 180,E1 -14315.923,E2 -14315.923} C_VEL
LIN {X 0,Y 340.443,Z 452.635,A -85,B 0,C 180,E1 -14318.308,E2 -14318.308} C_VEL
LIN {X 0,Y 340.603,Z 452.28,A -85,B 0,C 180,E1 -14320.701,E2 -14320.701} C_VEL
LIN {X 0,Y 340.778,Z 451.478,A -85,B 0,C 180,E1 -14321.901,E2 -14321.901} C_VEL
LIN {X 0,Y 341.026,Z 450.273,A -85,B 0,C 180,E1 -14323.102,E2 -14323.102} C_VEL
LIN {X 0,Y 341.527,Z 447.993,A -85,B 0,C 180,E1 -14324.719,E2 -14324.719} C_VEL
LIN {X 0,Y 342.287,Z 444.054,A -85,B 0,C 180,E1 -14326.705,E2 -14326.705} C_VEL
LIN {X 0,Y 343.103,Z 439.294,A -85,B 0,C 180,E1 -14328.511,E2 -14328.511} C_VEL
LIN {X 0,Y 344.17,Z 433.231,A -85,B 0,C 180,E1 -14330.312,E2 -14330.312} C_VEL
LIN {X 0,Y 345.446,Z 425.618,A -85,B 0,C 180,E1 -14332.109,E2 -14332.109} C_VEL
LIN {X 0,Y 346.611,Z 417.748,A -85,B 0,C 180,E1 -14333.606,E2 -14333.606} C_VEL
LIN {X 0,Y 347.864,Z 408.073,A -85,B 0,C 180,E1 -14335.103,E2 -14335.103} C_VEL
LIN {X 0,Y 349.131,Z 397.517,A -85,B 0,C 180,E1 -14336.412,E2 -14336.412} C_VEL
LIN {X 0,Y 349.984,Z 389.373,A -85,B 0,C 180,E1 -14337.229,E2 -14337.229} C_VEL
LIN {X 0,Y 347.588,Z 380.956,A -85,B 0,C 180,E1 -14338.19,E2 -14338.19} C_VEL
LIN {X 0,Y 343.464,Z 369.894,A -85,B 0,C 180,E1 -14339.328,E2 -14339.328} C_VEL
LIN {X 0,Y 340.828,Z 363.704,A -85,B 0,C 180,E1 -14339.903,E2 -14339.903} C_VEL
LIN {X 0,Y 340.732,Z 363.049,A -85,B 0,C 180,E1 -14339.967,E2 -14339.967} C_VEL
LIN {X 0,Y 340.692,Z 363.045,A -85,B 0,C 180,E1 -14343.846,E2 -14343.846} C_VEL
LIN {X 0,Y 340.705,Z 363.05,A -85,B 0,C 180,E1 -14346.74,E2 -14346.74} C_VEL
LIN {X 0,Y 340.688,Z 363.047,A -85,B 0,C 180,E1 -14350.246,E2 -14350.246} C_VEL
LIN {X 0,Y 340.652,Z 363.053,A -85,B 0,C 180,E1 -14353.772,E2 -14353.772} C_VEL
LIN {X 0,Y 340.73,Z 363.046,A -85,B 0,C 180,E1 -14357.948,E2 -14357.948} C_VEL
LIN {X 0,Y 340.71,Z 363.048,A -85,B 0,C 180,E1 -14361.502,E2 -14361.502} C_VEL
LIN {X 0,Y 340.082,Z 363.132,A -85,B 0,C 180,E1 -14362.488,E2 -14362.488} C_VEL
LIN {X 0,Y 337.196,Z 363.488,A -85,B 0,C 180,E1 -14364.092,E2 -14364.092} C_VEL
LIN {X 0,Y 334.738,Z 363.791,A -85,B 0,C 180,E1 -14365.391,E2 -14365.391} C_VEL
LIN {X 0,Y 333.706,Z 363.917,A -85,B 0,C 180,E1 -14366.397,E2 -14366.397} C_VEL
LIN {X 0,Y 333.637,Z 363.924,A -85,B 0,C 180,E1 -14366.738,E2 -14366.738} C_VEL
LIN {X 0,Y 333.702,Z 363.884,A -85,B 0,C 180,E1 -14369.709,E2 -14369.709} C_VEL
LIN {X 0,Y 333.742,Z 363.903,A -85,B 0,C 180,E1 -14372.401,E2 -14372.401} C_VEL
LIN {X 0,Y 333.724,Z 363.914,A -85,B 0,C 180,E1 -14375.09,E2 -14375.09} C_VEL
LIN {X 0,Y 333.684,Z 363.92,A -85,B 0,C 180,E1 -14379.019,E2 -14379.019} C_VEL
LIN {X 0,Y 333.791,Z 363.9,A -85,B 0,C 180,E1 -14381.589,E2 -14381.589} C_VEL
LIN {X 0,Y 333.805,Z 363.906,A -85,B 0,C 180,E1 -14385.576,E2 -14385.576} C_VEL
LIN {X 0,Y 333.835,Z 363.902,A -85,B 0,C 180,E1 -14389.078,E2 -14389.078} C_VEL
LIN {X 0,Y 334.022,Z 363.876,A -85,B 0,C 180,E1 -14392.747,E2 -14392.747} C_VEL
LIN {X 0,Y 333.81,Z 363.897,A -85,B 0,C 180,E1 -14395.169,E2 -14395.169} C_VEL
LIN {X 0,Y 334.129,Z 363.865,A -85,B 0,C 180,E1 -14397.589,E2 -14397.589} C_VEL
LIN {X 0,Y 334.264,Z 363.838,A -85,B 0,C 180,E1 -14400,E2 -14400} C_VEL
LIN {X 0,Y 334.128,Z 363.867,A -85,B 0,C 180,E1 -14402.411,E2 -14402.411} C_VEL
LIN {X 0,Y 334.022,Z 363.88,A -85,B 0,C 180,E1 -14407.252,E2 -14407.252} C_VEL
LIN {X 0,Y 333.83,Z 363.899,A -85,B 0,C 180,E1 -14410.922,E2 -14410.922} C_VEL
LIN {X 0,Y 333.804,Z 363.902,A -85,B 0,C 180,E1 -14414.634,E2 -14414.634} C_VEL
LIN {X 0,Y 333.793,Z 363.908,A -85,B 0,C 180,E1 -14418.656,E2 -14418.656} C_VEL
LIN {X 0,Y 333.688,Z 363.923,A -85,B 0,C 180,E1 -14422.278,E2 -14422.278} C_VEL
LIN {X 0,Y 333.732,Z 363.919,A -85,B 0,C 180,E1 -14426.246,E2 -14426.246} C_VEL
LIN {X 0,Y 333.708,Z 363.921,A -85,B 0,C 180,E1 -14428.972,E2 -14428.972} C_VEL
LIN {X 0,Y 333.642,Z 363.928,A -85,B 0,C 180,E1 -14432.588,E2 -14432.588} C_VEL
LIN {X 0,Y 333.674,Z 363.921,A -85,B 0,C 180,E1 -14436.139,E2 -14436.139} C_VEL
LIN {X 0,Y 333.681,Z 363.911,A -85,B 0,C 180,E1 -14439.187,E2 -14439.187} C_VEL
LIN {X 0,Y 333.697,Z 364.073,A -85,B 0,C 180,E1 -14441.159,E2 -14441.159} C_VEL
LIN {X 0,Y 335.014,Z 370.268,A -85,B 0,C 180,E1 -14444.501,E2 -14444.501} C_VEL
LIN {X 0,Y 336.387,Z 377.333,A -85,B 0,C 180,E1 -14448.045,E2 -14448.045} C_VEL
LIN {X 0,Y 337.677,Z 384.406,A -85,B 0,C 180,E1 -14451.364,E2 -14451.364} C_VEL
LIN {X 0,Y 337.906,Z 386.331,A -85,B 0,C 180,E1 -14452.218,E2 -14452.218} C_VEL
LIN {X 0,Y 337.183,Z 391.556,A -85,B 0,C 180,E1 -14454.379,E2 -14454.379} C_VEL
LIN {X 0,Y 335.975,Z 399.978,A -85,B 0,C 180,E1 -14457.765,E2 -14457.765} C_VEL
LIN {X 0,Y 334.7,Z 410.486,A -85,B 0,C 180,E1 -14461.874,E2 -14461.874} C_VEL
LIN {X 0,Y 333.787,Z 420.592,A -85,B 0,C 180,E1 -14465.76,E2 -14465.76} C_VEL
LIN {X 0,Y 333.5,Z 423.937,A -85,B 0,C 180,E1 -14467.002,E2 -14467.002} C_VEL
LIN {X 0,Y 336.183,Z 438.237,A -85,B 0,C 180,E1 -14467.737,E2 -14467.737} C_VEL
LIN {X 0,Y 337.89,Z 451.287,A -85,B 0,C 180,E1 -14468.609,E2 -14468.609} C_VEL
LIN {X 0,Y 338.697,Z 463.745,A -85,B 0,C 180,E1 -14469.639,E2 -14469.639} C_VEL
LIN {X 0,Y 338.643,Z 475.049,A -85,B 0,C 180,E1 -14470.765,E2 -14470.765} C_VEL
LIN {X 0,Y 338.067,Z 482.866,A -85,B 0,C 180,E1 -14471.675,E2 -14471.675} C_VEL
LIN {X 0,Y 336.502,Z 492.639,A -85,B 0,C 180,E1 -14472.999,E2 -14472.999} C_VEL
LIN {X 0,Y 335.15,Z 502.234,A -85,B 0,C 180,E1 -14474.613,E2 -14474.613} C_VEL
LIN {X 0,Y 334.072,Z 510.405,A -85,B 0,C 180,E1 -14476.311,E2 -14476.311} C_VEL
LIN {X 0,Y 333.198,Z 517.485,A -85,B 0,C 180,E1 -14478.133,E2 -14478.133} C_VEL
LIN {X 0,Y 332.615,Z 524.051,A -85,B 0,C 180,E1 -14480.269,E2 -14480.269} C_VEL
LIN {X 0,Y 332.457,Z 528.419,A -85,B 0,C 180,E1 -14482.103,E2 -14482.103} C_VEL
LIN {X 0,Y 332.531,Z 531.734,A -85,B 0,C 180,E1 -14483.935,E2 -14483.935} C_VEL
LIN {X 0,Y 332.598,Z 533.404,A -85,B 0,C 180,E1 -14485.152,E2 -14485.152} C_VEL
LIN {X 0,Y 332.785,Z 534.653,A -85,B 0,C 180,E1 -14486.368,E2 -14486.368} C_VEL
LIN {X 0,Y 332.867,Z 535.448,A -85,B 0,C 180,E1 -14487.581,E2 -14487.581} C_VEL
LIN {X 0,Y 332.967,Z 535.834,A -85,B 0,C 180,E1 -14490.001,E2 -14490.001} C_VEL
LIN {X 0,Y 332.924,Z 535.401,A -85,B 0,C 180,E1 -14491.21,E2 -14491.21} C_VEL
LIN {X 0,Y 332.921,Z 534.523,A -85,B 0,C 180,E1 -14492.421,E2 -14492.421} C_VEL
LIN {X 0,Y 332.968,Z 533.237,A -85,B 0,C 180,E1 -14493.631,E2 -14493.631} C_VEL
LIN {X 0,Y 332.689,Z 530.43,A -85,B 0,C 180,E1 -14495.456,E2 -14495.456} C_VEL
LIN {X 0,Y 332.613,Z 526.577,A -85,B 0,C 180,E1 -14497.284,E2 -14497.284} C_VEL
LIN {X 0,Y 332.631,Z 521.559,A -85,B 0,C 180,E1 -14499.119,E2 -14499.119} C_VEL
LIN {X 0,Y 332.883,Z 515.245,A -85,B 0,C 180,E1 -14500.954,E2 -14500.954} C_VEL
LIN {X 0,Y 333.495,Z 507.421,A -85,B 0,C 180,E1 -14502.785,E2 -14502.785} C_VEL
LIN {X 0,Y 334.197,Z 499.415,A -85,B 0,C 180,E1 -14504.307,E2 -14504.307} C_VEL
LIN {X 0,Y 335.336,Z 489.691,A -85,B 0,C 180,E1 -14505.811,E2 -14505.811} C_VEL
LIN {X 0,Y 336.321,Z 478.868,A -85,B 0,C 180,E1 -14507.168,E2 -14507.168} C_VEL
LIN {X 0,Y 336.519,Z 473.133,A -85,B 0,C 180,E1 -14507.785,E2 -14507.785} C_VEL
LIN {X 0,Y 336.158,Z 461.899,A -85,B 0,C 180,E1 -14508.824,E2 -14508.824} C_VEL
LIN {X 0,Y 335.415,Z 449.126,A -85,B 0,C 180,E1 -14509.748,E2 -14509.748} C_VEL
LIN {X 0,Y 334.263,Z 436.005,A -85,B 0,C 180,E1 -14510.461,E2 -14510.461} C_VEL
LIN {X 0,Y 332.963,Z 425.114,A -85,B 0,C 180,E1 -14510.908,E2 -14510.908} C_VEL
LIN {X 0,Y 333.663,Z 413.851,A -85,B 0,C 180,E1 -14515.08,E2 -14515.08} C_VEL
LIN {X 0,Y 334.476,Z 403.624,A -85,B 0,C 180,E1 -14518.901,E2 -14518.901} C_VEL
LIN {X 0,Y 335.361,Z 394.587,A -85,B 0,C 180,E1 -14522.304,E2 -14522.304} C_VEL
LIN {X 0,Y 336.651,Z 383.77,A -85,B 0,C 180,E1 -14526.512,E2 -14526.512} C_VEL
LIN {X 0,Y 336.781,Z 381.204,A -85,B 0,C 180,E1 -14527.534,E2 -14527.534} C_VEL
LIN {X 0,Y 335.703,Z 374.344,A -85,B 0,C 180,E1 -14530.467,E2 -14530.467} C_VEL
LIN {X 0,Y 334.042,Z 365.847,A -85,B 0,C 180,E1 -14534.329,E2 -14534.329} C_VEL
LIN {X 0,Y 333.689,Z 363.922,A -85,B 0,C 180,E1 -14535.263,E2 -14535.263} C_VEL
LIN {X 0,Y 333.651,Z 363.924,A -85,B 0,C 180,E1 -14539.316,E2 -14539.316} C_VEL
LIN {X 0,Y 333.669,Z 363.923,A -85,B 0,C 180,E1 -14543.168,E2 -14543.168} C_VEL
LIN {X 0,Y 333.678,Z 363.92,A -85,B 0,C 180,E1 -14545.342,E2 -14545.342} C_VEL
LIN {X 0,Y 333.695,Z 363.916,A -85,B 0,C 180,E1 -14549.638,E2 -14549.638} C_VEL
LIN {X 0,Y 333.744,Z 363.912,A -85,B 0,C 180,E1 -14552.401,E2 -14552.401} C_VEL
LIN {X 0,Y 333.732,Z 363.913,A -85,B 0,C 180,E1 -14555.091,E2 -14555.091} C_VEL
LIN {X 0,Y 333.69,Z 363.919,A -85,B 0,C 180,E1 -14559.02,E2 -14559.02} C_VEL
LIN {X 0,Y 333.799,Z 363.903,A -85,B 0,C 180,E1 -14561.59,E2 -14561.59} C_VEL
LIN {X 0,Y 333.814,Z 363.901,A -85,B 0,C 180,E1 -14565.577,E2 -14565.577} C_VEL
LIN {X 0,Y 333.839,Z 363.898,A -85,B 0,C 180,E1 -14569.078,E2 -14569.078} C_VEL
LIN {X 0,Y 334.032,Z 363.876,A -85,B 0,C 180,E1 -14572.748,E2 -14572.748} C_VEL
LIN {X 0,Y 333.814,Z 363.901,A -85,B 0,C 180,E1 -14575.169,E2 -14575.169} C_VEL
LIN {X 0,Y 334.111,Z 363.864,A -85,B 0,C 180,E1 -14577.589,E2 -14577.589} C_VEL
LIN {X 0,Y 334.253,Z 363.849,A -85,B 0,C 180,E1 -14580,E2 -14580} C_VEL
LIN {X 0,Y 334.111,Z 363.867,A -85,B 0,C 180,E1 -14582.411,E2 -14582.411} C_VEL
LIN {X 0,Y 334.032,Z 363.872,A -85,B 0,C 180,E1 -14587.253,E2 -14587.253} C_VEL
LIN {X 0,Y 333.84,Z 363.897,A -85,B 0,C 180,E1 -14590.922,E2 -14590.922} C_VEL
LIN {X 0,Y 333.814,Z 363.9,A -85,B 0,C 180,E1 -14594.634,E2 -14594.634} C_VEL
LIN {X 0,Y 333.803,Z 363.902,A -85,B 0,C 180,E1 -14598.656,E2 -14598.656} C_VEL
LIN {X 0,Y 333.698,Z 363.916,A -85,B 0,C 180,E1 -14602.278,E2 -14602.278} C_VEL
LIN {X 0,Y 333.741,Z 363.911,A -85,B 0,C 180,E1 -14606.246,E2 -14606.246} C_VEL
LIN {X 0,Y 333.71,Z 363.913,A -85,B 0,C 180,E1 -14610.29,E2 -14610.29} C_VEL
LIN {X 0,Y 333.68,Z 363.917,A -85,B 0,C 180,E1 -14614.659,E2 -14614.659} C_VEL
LIN {X 0,Y 333.66,Z 363.924,A -85,B 0,C 180,E1 -14617.651,E2 -14617.651} C_VEL
LIN {X 0,Y 333.653,Z 363.921,A -85,B 0,C 180,E1 -14620.767,E2 -14620.767} C_VEL
LIN {X 0,Y 333.63,Z 363.923,A -85,B 0,C 180,E1 -14624.256,E2 -14624.256} C_VEL
LIN {X 0,Y 333.648,Z 363.924,A -85,B 0,C 180,E1 -14627.618,E2 -14627.618} C_VEL
LIN {X 0,Y 333.658,Z 363.925,A -85,B 0,C 180,E1 -14631.202,E2 -14631.202} C_VEL
LIN {X 0,Y 333.682,Z 363.917,A -85,B 0,C 180,E1 -14633.861,E2 -14633.861} C_VEL
LIN {X 0,Y 333.649,Z 363.924,A -85,B 0,C 180,E1 -14637.413,E2 -14637.413} C_VEL
LIN {X 0,Y 333.717,Z 363.918,A -85,B 0,C 180,E1 -14641.027,E2 -14641.027} C_VEL
LIN {X 0,Y 333.742,Z 363.91,A -85,B 0,C 180,E1 -14643.753,E2 -14643.753} C_VEL
LIN {X 0,Y 333.725,Z 363.912,A -85,B 0,C 180,E1 -14647.913,E2 -14647.913} C_VEL
LIN {X 0,Y 333.799,Z 363.903,A -85,B 0,C 180,E1 -14651.589,E2 -14651.589} C_VEL
LIN {X 0,Y 333.814,Z 363.901,A -85,B 0,C 180,E1 -14655.576,E2 -14655.576} C_VEL
LIN {X 0,Y 333.816,Z 363.901,A -85,B 0,C 180,E1 -14657.884,E2 -14657.884} C_VEL
LIN {X 0,Y 337.861,Z 376.677,A -85,B 0,C 180,E1 -14658.936,E2 -14658.936} C_VEL
LIN {X 0,Y 340.158,Z 384.899,A -85,B 0,C 180,E1 -14659.737,E2 -14659.737} C_VEL
LIN {X 0,Y 339.225,Z 395.66,A -85,B 0,C 180,E1 -14660.76,E2 -14660.76} C_VEL
LIN {X 0,Y 338.267,Z 406.648,A -85,B 0,C 180,E1 -14662.088,E2 -14662.088} C_VEL
LIN {X 0,Y 337.404,Z 415.52,A -85,B 0,C 180,E1 -14663.421,E2 -14663.421} C_VEL
LIN {X 0,Y 336.372,Z 425.122,A -85,B 0,C 180,E1 -14665.205,E2 -14665.205} C_VEL
LIN {X 0,Y 335.43,Z 432.851,A -85,B 0,C 180,E1 -14666.997,E2 -14666.997} C_VEL
LIN {X 0,Y 334.707,Z 439.018,A -85,B 0,C 180,E1 -14668.796,E2 -14668.796} C_VEL
LIN {X 0,Y 334.167,Z 443.929,A -85,B 0,C 180,E1 -14670.602,E2 -14670.602} C_VEL
LIN {X 0,Y 333.7,Z 447.753,A -85,B 0,C 180,E1 -14672.413,E2 -14672.413} C_VEL
LIN {X 0,Y 333.474,Z 449.727,A -85,B 0,C 180,E1 -14673.624,E2 -14673.624} C_VEL
LIN {X 0,Y 333.473,Z 451.276,A -85,B 0,C 180,E1 -14674.835,E2 -14674.835} C_VEL
LIN {X 0,Y 333.437,Z 452.431,A -85,B 0,C 180,E1 -14676.049,E2 -14676.049} C_VEL
LIN {X 0,Y 333.41,Z 453.526,A -85,B 0,C 180,E1 -14678.484,E2 -14678.484} C_VEL
LIN {X 0,Y 333.472,Z 453.511,A -85,B 0,C 180,E1 -14679.706,E2 -14679.706} C_VEL
LIN {X 0,Y 333.591,Z 453.098,A -85,B 0,C 180,E1 -14680.929,E2 -14680.929} C_VEL
LIN {X 0,Y 334.083,Z 451.019,A -85,B 0,C 180,E1 -14683.379,E2 -14683.379} C_VEL
LIN {X 0,Y 334.57,Z 448.868,A -85,B 0,C 180,E1 -14684.92,E2 -14684.92} C_VEL
LIN {X 0,Y 335.423,Z 444.677,A -85,B 0,C 180,E1 -14687.057,E2 -14687.057} C_VEL
LIN {X 0,Y 336.316,Z 439.847,A -85,B 0,C 180,E1 -14688.898,E2 -14688.898} C_VEL
LIN {X 0,Y 337.448,Z 433.709,A -85,B 0,C 180,E1 -14690.735,E2 -14690.735} C_VEL
LIN {X 0,Y 338.81,Z 425.963,A -85,B 0,C 180,E1 -14692.565,E2 -14692.565} C_VEL
LIN {X 0,Y 340.04,Z 417.984,A -85,B 0,C 180,E1 -14694.091,E2 -14694.091} C_VEL
LIN {X 0,Y 341.357,Z 408.179,A -85,B 0,C 180,E1 -14695.616,E2 -14695.616} C_VEL
LIN {X 0,Y 342.584,Z 398.483,A -85,B 0,C 180,E1 -14696.828,E2 -14696.828} C_VEL
LIN {X 0,Y 343.385,Z 390.909,A -85,B 0,C 180,E1 -14697.61,E2 -14697.61} C_VEL
LIN {X 0,Y 340.49,Z 381.321,A -85,B 0,C 180,E1 -14698.749,E2 -14698.749} C_VEL
LIN {X 0,Y 336.388,Z 370.67,A -85,B 0,C 180,E1 -14699.884,E2 -14699.884} C_VEL
LIN {X 0,Y 333.792,Z 364.657,A -85,B 0,C 180,E1 -14700.464,E2 -14700.464} C_VEL
LIN {X 0,Y 333.679,Z 363.923,A -85,B 0,C 180,E1 -14700.553,E2 -14700.553} C_VEL
LIN {X 0,Y 333.686,Z 363.923,A -85,B 0,C 180,E1 -14704.773,E2 -14704.773} C_VEL
LIN {X 0,Y 333.652,Z 363.925,A -85,B 0,C 180,E1 -14707.65,E2 -14707.65} C_VEL
LIN {X 0,Y 333.646,Z 363.927,A -85,B 0,C 180,E1 -14710.766,E2 -14710.766} C_VEL
LIN {X 0,Y 333.594,Z 363.931,A -85,B 0,C 180,E1 -14714.25,E2 -14714.25} C_VEL
LIN {X 0,Y 333.672,Z 363.923,A -85,B 0,C 180,E1 -14717.623,E2 -14717.623} C_VEL
LIN {X 0,Y 333.659,Z 363.924,A -85,B 0,C 180,E1 -14721.492,E2 -14721.492} C_VEL
LIN {X 0,Y 333.672,Z 363.924,A -85,B 0,C 180,E1 -14725.341,E2 -14725.341} C_VEL
LIN {X 0,Y 333.637,Z 363.924,A -85,B 0,C 180,E1 -14726.738,E2 -14726.738} C_VEL
LIN {X 0,Y 333.015,Z 364.004,A -85,B 0,C 180,E1 -14727.746,E2 -14727.746} C_VEL
LIN {X 0,Y 330.2,Z 364.348,A -85,B 0,C 180,E1 -14729.388,E2 -14729.388} C_VEL
LIN {X 0,Y 327.786,Z 364.64,A -85,B 0,C 180,E1 -14730.717,E2 -14730.717} C_VEL
LIN {X 0,Y 326.741,Z 364.769,A -85,B 0,C 180,E1 -14731.746,E2 -14731.746} C_VEL
LIN {X 0,Y 326.652,Z 364.781,A -85,B 0,C 180,E1 -14732.094,E2 -14732.094} C_VEL
LIN {X 0,Y 326.685,Z 364.791,A -85,B 0,C 180,E1 -14734.626,E2 -14734.626} C_VEL
LIN {X 0,Y 326.646,Z 364.795,A -85,B 0,C 180,E1 -14738.545,E2 -14738.545} C_VEL
LIN {X 0,Y 326.741,Z 364.78,A -85,B 0,C 180,E1 -14741.177,E2 -14741.177} C_VEL
LIN {X 0,Y 326.759,Z 364.784,A -85,B 0,C 180,E1 -14745.432,E2 -14745.432} C_VEL
LIN {X 0,Y 326.771,Z 364.782,A -85,B 0,C 180,E1 -14748.839,E2 -14748.839} C_VEL
LIN {X 0,Y 326.976,Z 364.754,A -85,B 0,C 180,E1 -14752.59,E2 -14752.59} C_VEL
LIN {X 0,Y 326.777,Z 364.772,A -85,B 0,C 180,E1 -14755.065,E2 -14755.065} C_VEL
LIN {X 0,Y 327.065,Z 364.745,A -85,B 0,C 180,E1 -14757.537,E2 -14757.537} C_VEL
LIN {X 0,Y 327.215,Z 364.715,A -85,B 0,C 180,E1 -14760,E2 -14760} C_VEL
LIN {X 0,Y 327.065,Z 364.747,A -85,B 0,C 180,E1 -14762.463,E2 -14762.463} C_VEL
LIN {X 0,Y 326.993,Z 364.75,A -85,B 0,C 180,E1 -14766.169,E2 -14766.169} C_VEL
LIN {X 0,Y 326.91,Z 364.762,A -85,B 0,C 180,E1 -14768.655,E2 -14768.655} C_VEL
LIN {X 0,Y 326.731,Z 364.786,A -85,B 0,C 180,E1 -14772.421,E2 -14772.421} C_VEL
LIN {X 0,Y 326.75,Z 364.782,A -85,B 0,C 180,E1 -14774.958,E2 -14774.958} C_VEL
LIN {X 0,Y 326.729,Z 364.787,A -85,B 0,C 180,E1 -14778.839,E2 -14778.839} C_VEL
LIN {X 0,Y 326.616,Z 364.803,A -85,B 0,C 180,E1 -14782.787,E2 -14782.787} C_VEL
LIN {X 0,Y 326.686,Z 364.796,A -85,B 0,C 180,E1 -14785.484,E2 -14785.484} C_VEL
LIN {X 0,Y 326.657,Z 364.799,A -85,B 0,C 180,E1 -14789.659,E2 -14789.659} C_VEL
LIN {X 0,Y 326.604,Z 364.804,A -85,B 0,C 180,E1 -14794.02,E2 -14794.02} C_VEL
LIN {X 0,Y 326.627,Z 364.798,A -85,B 0,C 180,E1 -14797.24,E2 -14797.24} C_VEL
LIN {X 0,Y 326.693,Z 364.983,A -85,B 0,C 180,E1 -14800.578,E2 -14800.578} C_VEL
LIN {X 0,Y 328.019,Z 371.356,A -85,B 0,C 180,E1 -14804.133,E2 -14804.133} C_VEL
LIN {X 0,Y 329.279,Z 377.861,A -85,B 0,C 180,E1 -14807.496,E2 -14807.496} C_VEL
LIN {X 0,Y 330.675,Z 385.48,A -85,B 0,C 180,E1 -14811.158,E2 -14811.158} C_VEL
LIN {X 0,Y 330.82,Z 389.002,A -85,B 0,C 180,E1 -14812.739,E2 -14812.739} C_VEL
LIN {X 0,Y 329.213,Z 399.318,A -85,B 0,C 180,E1 -14817.019,E2 -14817.019} C_VEL
LIN {X 0,Y 327.877,Z 409.401,A -85,B 0,C 180,E1 -14821.079,E2 -14821.079} C_VEL
LIN {X 0,Y 326.812,Z 419.866,A -85,B 0,C 180,E1 -14825.208,E2 -14825.208} C_VEL
LIN {X 0,Y 326.536,Z 422.886,A -85,B 0,C 180,E1 -14826.395,E2 -14826.395} C_VEL
LIN {X 0,Y 329.309,Z 437.345,A -85,B 0,C 180,E1 -14827.175,E2 -14827.175} C_VEL
LIN {X 0,Y 331.063,Z 450.677,A -85,B 0,C 180,E1 -14828.097,E2 -14828.097} C_VEL
LIN {X 0,Y 331.87,Z 463.119,A -85,B 0,C 180,E1 -14829.158,E2 -14829.158} C_VEL
LIN {X 0,Y 331.837,Z 474.749,A -85,B 0,C 180,E1 -14830.354,E2 -14830.354} C_VEL
LIN {X 0,Y 331.279,Z 482.463,A -85,B 0,C 180,E1 -14831.285,E2 -14831.285} C_VEL
LIN {X 0,Y 329.697,Z 492.153,A -85,B 0,C 180,E1 -14832.638,E2 -14832.638} C_VEL
LIN {X 0,Y 328.379,Z 500.738,A -85,B 0,C 180,E1 -14834.107,E2 -14834.107} C_VEL
LIN {X 0,Y 327.408,Z 508.436,A -85,B 0,C 180,E1 -14835.71,E2 -14835.71} C_VEL
LIN {X 0,Y 326.472,Z 514.608,A -85,B 0,C 180,E1 -14837.254,E2 -14837.254} C_VEL
LIN {X 0,Y 325.648,Z 521.643,A -85,B 0,C 180,E1 -14839.431,E2 -14839.431} C_VEL
LIN {X 0,Y 325.407,Z 526.35,A -85,B 0,C 180,E1 -14841.305,E2 -14841.305} C_VEL
LIN {X 0,Y 325.407,Z 530.41,A -85,B 0,C 180,E1 -14843.458,E2 -14843.458} C_VEL
LIN {X 0,Y 325.514,Z 532.594,A -85,B 0,C 180,E1 -14845.047,E2 -14845.047} C_VEL
LIN {X 0,Y 325.714,Z 533.814,A -85,B 0,C 180,E1 -14846.289,E2 -14846.289} C_VEL
LIN {X 0,Y 325.818,Z 534.597,A -85,B 0,C 180,E1 -14847.528,E2 -14847.528} C_VEL
LIN {X 0,Y 325.92,Z 534.953,A -85,B 0,C 180,E1 -14850.001,E2 -14850.001} C_VEL
LIN {X 0,Y 325.877,Z 534.491,A -85,B 0,C 180,E1 -14851.237,E2 -14851.237} C_VEL
LIN {X 0,Y 325.876,Z 533.595,A -85,B 0,C 180,E1 -14852.473,E2 -14852.473} C_VEL
LIN {X 0,Y 325.887,Z 532.288,A -85,B 0,C 180,E1 -14853.71,E2 -14853.71} C_VEL
LIN {X 0,Y 325.62,Z 529.447,A -85,B 0,C 180,E1 -14855.575,E2 -14855.575} C_VEL
LIN {X 0,Y 325.534,Z 525.554,A -85,B 0,C 180,E1 -14857.444,E2 -14857.444} C_VEL
LIN {X 0,Y 325.566,Z 520.495,A -85,B 0,C 180,E1 -14859.318,E2 -14859.318} C_VEL
LIN {X 0,Y 325.87,Z 514.139,A -85,B 0,C 180,E1 -14861.193,E2 -14861.193} C_VEL
LIN {X 0,Y 326.479,Z 506.241,A -85,B 0,C 180,E1 -14863.064,E2 -14863.064} C_VEL
LIN {X 0,Y 327.159,Z 498.794,A -85,B 0,C 180,E1 -14864.51,E2 -14864.51} C_VEL
LIN {X 0,Y 328.455,Z 488.376,A -85,B 0,C 180,E1 -14866.151,E2 -14866.151} C_VEL
LIN {X 0,Y 329.533,Z 477.473,A -85,B 0,C 180,E1 -14867.533,E2 -14867.533} C_VEL
LIN {X 0,Y 329.359,Z 466.646,A -85,B 0,C 180,E1 -14868.668,E2 -14868.668} C_VEL
LIN {X 0,Y 328.793,Z 454.613,A -85,B 0,C 180,E1 -14869.677,E2 -14869.677} C_VEL
LIN {X 0,Y 327.864,Z 440.948,A -85,B 0,C 180,E1 -14870.55,E2 -14870.55} C_VEL
LIN {X 0,Y 326.352,Z 427.806,A -85,B 0,C 180,E1 -14871.16,E2 -14871.16} C_VEL
LIN {X 0,Y 325.942,Z 424.334,A -85,B 0,C 180,E1 -14871.276,E2 -14871.276} C_VEL
LIN {X 0,Y 326.64,Z 413.238,A -85,B 0,C 180,E1 -14875.489,E2 -14875.489} C_VEL
LIN {X 0,Y 327.575,Z 402.608,A -85,B 0,C 180,E1 -14879.569,E2 -14879.569} C_VEL
LIN {X 0,Y 328.459,Z 393.989,A -85,B 0,C 180,E1 -14882.918,E2 -14882.918} C_VEL
LIN {X 0,Y 329.653,Z 384.607,A -85,B 0,C 180,E1 -14886.652,E2 -14886.652} C_VEL
LIN {X 0,Y 329.7,Z 381.476,A -85,B 0,C 180,E1 -14887.935,E2 -14887.935} C_VEL
LIN {X 0,Y 328.664,Z 375.308,A -85,B 0,C 180,E1 -14890.662,E2 -14890.662} C_VEL
LIN {X 0,Y 327.22,Z 367.908,A -85,B 0,C 180,E1 -14894.088,E2 -14894.088} C_VEL
LIN {X 0,Y 326.589,Z 364.806,A -85,B 0,C 180,E1 -14895.675,E2 -14895.675} C_VEL
LIN {X 0,Y 326.595,Z 364.8,A -85,B 0,C 180,E1 -14899.792,E2 -14899.792} C_VEL
LIN {X 0,Y 326.634,Z 364.801,A -85,B 0,C 180,E1 -14902.954,E2 -14902.954} C_VEL
LIN {X 0,Y 326.611,Z 364.799,A -85,B 0,C 180,E1 -14905.981,E2 -14905.981} C_VEL
LIN {X 0,Y 326.652,Z 364.795,A -85,B 0,C 180,E1 -14910.34,E2 -14910.34} C_VEL
LIN {X 0,Y 326.695,Z 364.792,A -85,B 0,C 180,E1 -14914.517,E2 -14914.517} C_VEL
LIN {X 0,Y 326.653,Z 364.798,A -85,B 0,C 180,E1 -14918.546,E2 -14918.546} C_VEL
LIN {X 0,Y 326.749,Z 364.782,A -85,B 0,C 180,E1 -14921.178,E2 -14921.178} C_VEL
LIN {X 0,Y 326.768,Z 364.779,A -85,B 0,C 180,E1 -14925.433,E2 -14925.433} C_VEL
LIN {X 0,Y 326.775,Z 364.78,A -85,B 0,C 180,E1 -14928.839,E2 -14928.839} C_VEL
LIN {X 0,Y 326.983,Z 364.755,A -85,B 0,C 180,E1 -14932.591,E2 -14932.591} C_VEL
LIN {X 0,Y 326.782,Z 364.777,A -85,B 0,C 180,E1 -14935.065,E2 -14935.065} C_VEL
LIN {X 0,Y 327.051,Z 364.742,A -85,B 0,C 180,E1 -14937.537,E2 -14937.537} C_VEL
LIN {X 0,Y 327.205,Z 364.726,A -85,B 0,C 180,E1 -14940,E2 -14940} C_VEL
LIN {X 0,Y 327.051,Z 364.746,A -85,B 0,C 180,E1 -14942.464,E2 -14942.464} C_VEL
LIN {X 0,Y 326.977,Z 364.751,A -85,B 0,C 180,E1 -14946.681,E2 -14946.681} C_VEL
LIN {X 0,Y 326.82,Z 364.776,A -85,B 0,C 180,E1 -14949.906,E2 -14949.906} C_VEL
LIN {X 0,Y 326.765,Z 364.781,A -85,B 0,C 180,E1 -14953.685,E2 -14953.685} C_VEL
LIN {X 0,Y 326.706,Z 364.788,A -85,B 0,C 180,E1 -14957.528,E2 -14957.528} C_VEL
LIN {X 0,Y 326.671,Z 364.793,A -85,B 0,C 180,E1 -14960.135,E2 -14960.135} C_VEL
LIN {X 0,Y 326.658,Z 364.794,A -85,B 0,C 180,E1 -14964.129,E2 -14964.129} C_VEL
LIN {X 0,Y 326.689,Z 364.788,A -85,B 0,C 180,E1 -14966.858,E2 -14966.858} C_VEL
LIN {X 0,Y 326.646,Z 364.792,A -85,B 0,C 180,E1 -14970.611,E2 -14970.611} C_VEL
LIN {X 0,Y 326.613,Z 364.799,A -85,B 0,C 180,E1 -14974.019,E2 -14974.019} C_VEL
LIN {X 0,Y 326.635,Z 364.798,A -85,B 0,C 180,E1 -14977.239,E2 -14977.239} C_VEL
LIN {X 0,Y 326.584,Z 364.804,A -85,B 0,C 180,E1 -14981.131,E2 -14981.131} C_VEL
LIN {X 0,Y 326.561,Z 364.804,A -85,B 0,C 180,E1 -14984.748,E2 -14984.748} C_VEL
LIN {X 0,Y 326.582,Z 364.801,A -85,B 0,C 180,E1 -14988.154,E2 -14988.154} C_VEL
LIN {X 0,Y 326.629,Z 364.799,A -85,B 0,C 180,E1 -14991.391,E2 -14991.391} C_VEL
LIN {X 0,Y 326.625,Z 364.799,A -85,B 0,C 180,E1 -14994.851,E2 -14994.851} C_VEL
LIN {X 0,Y 326.614,Z 364.8,A -85,B 0,C 180,E1 -14997.455,E2 -14997.455} C_VEL
LIN {X 0,Y 326.666,Z 364.792,A -85,B 0,C 180,E1 -15000.341,E2 -15000.341} C_VEL
LIN {X 0,Y 326.696,Z 364.789,A -85,B 0,C 180,E1 -15004.516,E2 -15004.516} C_VEL
LIN {X 0,Y 326.654,Z 364.795,A -85,B 0,C 180,E1 -15008.545,E2 -15008.545} C_VEL
LIN {X 0,Y 326.75,Z 364.784,A -85,B 0,C 180,E1 -15011.177,E2 -15011.177} C_VEL
LIN {X 0,Y 326.769,Z 364.78,A -85,B 0,C 180,E1 -15015.432,E2 -15015.432} C_VEL
LIN {X 0,Y 326.765,Z 364.78,A -85,B 0,C 180,E1 -15017.5,E2 -15017.5} C_VEL
LIN {X 0,Y 331.066,Z 378.248,A -85,B 0,C 180,E1 -15018.644,E2 -15018.644} C_VEL
LIN {X 0,Y 333.332,Z 386.414,A -85,B 0,C 180,E1 -15019.471,E2 -15019.471} C_VEL
LIN {X 0,Y 332.344,Z 397.528,A -85,B 0,C 180,E1 -15020.567,E2 -15020.567} C_VEL
LIN {X 0,Y 331.333,Z 408.269,A -85,B 0,C 180,E1 -15021.921,E2 -15021.921} C_VEL
LIN {X 0,Y 330.296,Z 418.754,A -85,B 0,C 180,E1 -15023.585,E2 -15023.585} C_VEL
LIN {X 0,Y 329.378,Z 426.514,A -85,B 0,C 180,E1 -15025.103,E2 -15025.103} C_VEL
LIN {X 0,Y 328.409,Z 434.117,A -85,B 0,C 180,E1 -15026.932,E2 -15026.932} C_VEL
LIN {X 0,Y 327.67,Z 440.206,A -85,B 0,C 180,E1 -15028.77,E2 -15028.77} C_VEL
LIN {X 0,Y 327.12,Z 445.05,A -85,B 0,C 180,E1 -15030.615,E2 -15030.615} C_VEL
LIN {X 0,Y 326.634,Z 448.814,A -85,B 0,C 180,E1 -15032.465,E2 -15032.465} C_VEL
LIN {X 0,Y 326.426,Z 450.757,A -85,B 0,C 180,E1 -15033.702,E2 -15033.702} C_VEL
LIN {X 0,Y 326.439,Z 452.275,A -85,B 0,C 180,E1 -15034.939,E2 -15034.939} C_VEL
LIN {X 0,Y 326.399,Z 453.375,A -85,B 0,C 180,E1 -15036.18,E2 -15036.18} C_VEL
LIN {X 0,Y 326.369,Z 454.418,A -85,B 0,C 180,E1 -15038.669,E2 -15038.669} C_VEL
LIN {X 0,Y 326.461,Z 454.373,A -85,B 0,C 180,E1 -15039.916,E2 -15039.916} C_VEL
LIN {X 0,Y 326.597,Z 453.904,A -85,B 0,C 180,E1 -15041.166,E2 -15041.166} C_VEL
LIN {X 0,Y 327.15,Z 451.767,A -85,B 0,C 180,E1 -15043.668,E2 -15043.668} C_VEL
LIN {X 0,Y 327.611,Z 449.754,A -85,B 0,C 180,E1 -15045.124,E2 -15045.124} C_VEL
LIN {X 0,Y 328.559,Z 445.304,A -85,B 0,C 180,E1 -15047.425,E2 -15047.425} C_VEL
LIN {X 0,Y 329.541,Z 440.403,A -85,B 0,C 180,E1 -15049.302,E2 -15049.302} C_VEL
LIN {X 0,Y 330.726,Z 434.183,A -85,B 0,C 180,E1 -15051.176,E2 -15051.176} C_VEL
LIN {X 0,Y 332.17,Z 426.308,A -85,B 0,C 180,E1 -15053.042,E2 -15053.042} C_VEL
LIN {X 0,Y 333.491,Z 418.221,A -85,B 0,C 180,E1 -15054.595,E2 -15054.595} C_VEL
LIN {X 0,Y 334.867,Z 408.286,A -85,B 0,C 180,E1 -15056.15,E2 -15056.15} C_VEL
LIN {X 0,Y 336.141,Z 398.391,A -85,B 0,C 180,E1 -15057.384,E2 -15057.384} C_VEL
LIN {X 0,Y 336.772,Z 393.094,A -85,B 0,C 180,E1 -15057.94,E2 -15057.94} C_VEL
LIN {X 0,Y 334.47,Z 384.869,A -85,B 0,C 180,E1 -15058.965,E2 -15058.965} C_VEL
LIN {X 0,Y 330.545,Z 374.358,A -85,B 0,C 180,E1 -15060.163,E2 -15060.163} C_VEL
LIN {X 0,Y 326.685,Z 365.183,A -85,B 0,C 180,E1 -15061.084,E2 -15061.084} C_VEL
LIN {X 0,Y 326.619,Z 364.801,A -85,B 0,C 180,E1 -15061.136,E2 -15061.136} C_VEL
LIN {X 0,Y 326.62,Z 364.805,A -85,B 0,C 180,E1 -15065.148,E2 -15065.148} C_VEL
LIN {X 0,Y 326.623,Z 364.802,A -85,B 0,C 180,E1 -15068.607,E2 -15068.607} C_VEL
LIN {X 0,Y 326.575,Z 364.804,A -85,B 0,C 180,E1 -15071.845,E2 -15071.845} C_VEL
LIN {X 0,Y 326.533,Z 364.813,A -85,B 0,C 180,E1 -15075.255,E2 -15075.255} C_VEL
LIN {X 0,Y 326.591,Z 364.807,A -85,B 0,C 180,E1 -15078.865,E2 -15078.865} C_VEL
LIN {X 0,Y 326.642,Z 364.8,A -85,B 0,C 180,E1 -15081.393,E2 -15081.393} C_VEL
LIN {X 0,Y 326.618,Z 364.801,A -85,B 0,C 180,E1 -15084.85,E2 -15084.85} C_VEL
LIN {X 0,Y 326.613,Z 364.793,A -85,B 0,C 180,E1 -15087.456,E2 -15087.456} C_VEL
LIN {X 0,Y 326.659,Z 364.761,A -85,B 0,C 180,E1 -15090.34,E2 -15090.34} C_VEL
LIN {X 0,Y 326.652,Z 364.781,A -85,B 0,C 180,E1 -15092.094,E2 -15092.094} C_VEL
LIN {X 0,Y 325.981,Z 364.875,A -85,B 0,C 180,E1 -15093.123,E2 -15093.123} C_VEL
LIN {X 0,Y 323.147,Z 365.232,A -85,B 0,C 180,E1 -15094.797,E2 -15094.797} C_VEL
LIN {X 0,Y 320.74,Z 365.525,A -85,B 0,C 180,E1 -15096.154,E2 -15096.154} C_VEL
LIN {X 0,Y 319.694,Z 365.652,A -85,B 0,C 180,E1 -15097.204,E2 -15097.204} C_VEL
LIN {X 0,Y 319.601,Z 365.665,A -85,B 0,C 180,E1 -15097.56,E2 -15097.56} C_VEL
LIN {X 0,Y 319.686,Z 365.661,A -85,B 0,C 180,E1 -15100.961,E2 -15100.961} C_VEL
LIN {X 0,Y 319.727,Z 365.661,A -85,B 0,C 180,E1 -15105.275,E2 -15105.275} C_VEL
LIN {X 0,Y 319.756,Z 365.652,A -85,B 0,C 180,E1 -15109.872,E2 -15109.872} C_VEL
LIN {X 0,Y 319.93,Z 365.632,A -85,B 0,C 180,E1 -15112.426,E2 -15112.426} C_VEL
LIN {X 0,Y 319.746,Z 365.646,A -85,B 0,C 180,E1 -15114.956,E2 -15114.956} C_VEL
LIN {X 0,Y 320.006,Z 365.625,A -85,B 0,C 180,E1 -15117.482,E2 -15117.482} C_VEL
LIN {X 0,Y 320.166,Z 365.593,A -85,B 0,C 180,E1 -15120,E2 -15120} C_VEL
LIN {X 0,Y 320.005,Z 365.626,A -85,B 0,C 180,E1 -15122.517,E2 -15122.517} C_VEL
LIN {X 0,Y 319.948,Z 365.628,A -85,B 0,C 180,E1 -15126.305,E2 -15126.305} C_VEL
LIN {X 0,Y 319.838,Z 365.642,A -85,B 0,C 180,E1 -15128.848,E2 -15128.848} C_VEL
LIN {X 0,Y 319.678,Z 365.664,A -85,B 0,C 180,E1 -15132.7,E2 -15132.7} C_VEL
LIN {X 0,Y 319.695,Z 365.662,A -85,B 0,C 180,E1 -15135.296,E2 -15135.296} C_VEL
LIN {X 0,Y 319.67,Z 365.668,A -85,B 0,C 180,E1 -15139.255,E2 -15139.255} C_VEL
LIN {X 0,Y 319.566,Z 365.678,A -85,B 0,C 180,E1 -15143.32,E2 -15143.32} C_VEL
LIN {X 0,Y 319.631,Z 365.675,A -85,B 0,C 180,E1 -15146.088,E2 -15146.088} C_VEL
LIN {X 0,Y 319.586,Z 365.68,A -85,B 0,C 180,E1 -15148.934,E2 -15148.934} C_VEL
LIN {X 0,Y 319.53,Z 365.686,A -85,B 0,C 180,E1 -15151.862,E2 -15151.862} C_VEL
LIN {X 0,Y 319.577,Z 365.676,A -85,B 0,C 180,E1 -15155.544,E2 -15155.544} C_VEL
LIN {X 0,Y 319.597,Z 365.665,A -85,B 0,C 180,E1 -15158.005,E2 -15158.005} C_VEL
LIN {X 0,Y 319.616,Z 365.814,A -85,B 0,C 180,E1 -15159.915,E2 -15159.915} C_VEL
LIN {X 0,Y 320.993,Z 372.441,A -85,B 0,C 180,E1 -15163.738,E2 -15163.738} C_VEL
LIN {X 0,Y 322.383,Z 379.506,A -85,B 0,C 180,E1 -15167.485,E2 -15167.485} C_VEL
LIN {X 0,Y 323.69,Z 386.594,A -85,B 0,C 180,E1 -15170.977,E2 -15170.977} C_VEL
LIN {X 0,Y 323.864,Z 390.086,A -85,B 0,C 180,E1 -15172.584,E2 -15172.584} C_VEL
LIN {X 0,Y 322.204,Z 400.379,A -85,B 0,C 180,E1 -15176.955,E2 -15176.955} C_VEL
LIN {X 0,Y 320.766,Z 410.672,A -85,B 0,C 180,E1 -15181.211,E2 -15181.211} C_VEL
LIN {X 0,Y 319.616,Z 421.872,A -85,B 0,C 180,E1 -15185.739,E2 -15185.739} C_VEL
LIN {X 0,Y 322.617,Z 437.828,A -85,B 0,C 180,E1 -15186.669,E2 -15186.669} C_VEL
LIN {X 0,Y 324.179,Z 449.405,A -85,B 0,C 180,E1 -15187.507,E2 -15187.507} C_VEL
LIN {X 0,Y 325.085,Z 461.973,A -85,B 0,C 180,E1 -15188.609,E2 -15188.609} C_VEL
LIN {X 0,Y 325.083,Z 473.01,A -85,B 0,C 180,E1 -15189.764,E2 -15189.764} C_VEL
LIN {X 0,Y 324.539,Z 482.062,A -85,B 0,C 180,E1 -15190.882,E2 -15190.882} C_VEL
LIN {X 0,Y 322.904,Z 491.67,A -85,B 0,C 180,E1 -15192.26,E2 -15192.26} C_VEL
LIN {X 0,Y 321.465,Z 500.398,A -85,B 0,C 180,E1 -15193.798,E2 -15193.798} C_VEL
LIN {X 0,Y 320.261,Z 509.138,A -85,B 0,C 180,E1 -15195.708,E2 -15195.708} C_VEL
LIN {X 0,Y 319.195,Z 516.115,A -85,B 0,C 180,E1 -15197.605,E2 -15197.605} C_VEL
LIN {X 0,Y 318.491,Z 522.598,A -85,B 0,C 180,E1 -15199.833,E2 -15199.833} C_VEL
LIN {X 0,Y 318.298,Z 526.893,A -85,B 0,C 180,E1 -15201.749,E2 -15201.749} C_VEL
LIN {X 0,Y 318.362,Z 530.143,A -85,B 0,C 180,E1 -15203.664,E2 -15203.664} C_VEL
LIN {X 0,Y 318.432,Z 531.781,A -85,B 0,C 180,E1 -15204.936,E2 -15204.936} C_VEL
LIN {X 0,Y 318.644,Z 532.974,A -85,B 0,C 180,E1 -15206.207,E2 -15206.207} C_VEL
LIN {X 0,Y 318.769,Z 533.746,A -85,B 0,C 180,E1 -15207.474,E2 -15207.474} C_VEL
LIN {X 0,Y 318.874,Z 534.072,A -85,B 0,C 180,E1 -15210.001,E2 -15210.001} C_VEL
LIN {X 0,Y 318.83,Z 533.579,A -85,B 0,C 180,E1 -15211.264,E2 -15211.264} C_VEL
LIN {X 0,Y 318.831,Z 532.667,A -85,B 0,C 180,E1 -15212.528,E2 -15212.528} C_VEL
LIN {X 0,Y 318.809,Z 531.338,A -85,B 0,C 180,E1 -15213.793,E2 -15213.793} C_VEL
LIN {X 0,Y 318.557,Z 528.464,A -85,B 0,C 180,E1 -15215.699,E2 -15215.699} C_VEL
LIN {X 0,Y 318.463,Z 524.53,A -85,B 0,C 180,E1 -15217.61,E2 -15217.61} C_VEL
LIN {X 0,Y 318.527,Z 519.431,A -85,B 0,C 180,E1 -15219.526,E2 -15219.526} C_VEL
LIN {X 0,Y 318.869,Z 513.031,A -85,B 0,C 180,E1 -15221.442,E2 -15221.442} C_VEL
LIN {X 0,Y 319.505,Z 505.052,A -85,B 0,C 180,E1 -15223.355,E2 -15223.355} C_VEL
LIN {X 0,Y 320.202,Z 497.272,A -85,B 0,C 180,E1 -15224.88,E2 -15224.88} C_VEL
LIN {X 0,Y 321.535,Z 487.039,A -85,B 0,C 180,E1 -15226.509,E2 -15226.509} C_VEL
LIN {X 0,Y 322.541,Z 476.011,A -85,B 0,C 180,E1 -15227.926,E2 -15227.926} C_VEL
LIN {X 0,Y 322.28,Z 463.808,A -85,B 0,C 180,E1 -15229.199,E2 -15229.199} C_VEL
LIN {X 0,Y 321.702,Z 451.752,A -85,B 0,C 180,E1 -15230.196,E2 -15230.196} C_VEL
LIN {X 0,Y 320.709,Z 438.613,A -85,B 0,C 180,E1 -15231.03,E2 -15231.03} C_VEL
LIN {X 0,Y 319.073,Z 425.237,A -85,B 0,C 180,E1 -15231.635,E2 -15231.635} C_VEL
LIN {X 0,Y 318.898,Z 423.312,A -85,B 0,C 180,E1 -15231.749,E2 -15231.749} C_VEL
LIN {X 0,Y 319.657,Z 412.201,A -85,B 0,C 180,E1 -15236.087,E2 -15236.087} C_VEL
LIN {X 0,Y 320.499,Z 403.367,A -85,B 0,C 180,E1 -15239.564,E2 -15239.564} C_VEL
LIN {X 0,Y 321.451,Z 394.436,A -85,B 0,C 180,E1 -15243.134,E2 -15243.134} C_VEL
LIN {X 0,Y 322.676,Z 385.336,A -85,B 0,C 180,E1 -15246.842,E2 -15246.842} C_VEL
LIN {X 0,Y 322.586,Z 381.808,A -85,B 0,C 180,E1 -15248.343,E2 -15248.343} C_VEL
LIN {X 0,Y 321.38,Z 374.966,A -85,B 0,C 180,E1 -15251.449,E2 -15251.449} C_VEL
LIN {X 0,Y 320.098,Z 368.349,A -85,B 0,C 180,E1 -15254.636,E2 -15254.636} C_VEL
LIN {X 0,Y 319.552,Z 365.684,A -85,B 0,C 180,E1 -15256.046,E2 -15256.046} C_VEL
LIN {X 0,Y 319.562,Z 365.677,A -85,B 0,C 180,E1 -15260.332,E2 -15260.332} C_VEL
LIN {X 0,Y 319.584,Z 365.676,A -85,B 0,C 180,E1 -15264.458,E2 -15264.458} C_VEL
LIN {X 0,Y 319.535,Z 365.68,A -85,B 0,C 180,E1 -15268.139,E2 -15268.139} C_VEL
LIN {X 0,Y 319.615,Z 365.67,A -85,B 0,C 180,E1 -15271.591,E2 -15271.591} C_VEL
LIN {X 0,Y 319.61,Z 365.672,A -85,B 0,C 180,E1 -15275.305,E2 -15275.305} C_VEL
LIN {X 0,Y 319.603,Z 365.673,A -85,B 0,C 180,E1 -15278.048,E2 -15278.048} C_VEL
LIN {X 0,Y 319.694,Z 365.663,A -85,B 0,C 180,E1 -15280.963,E2 -15280.963} C_VEL
LIN {X 0,Y 319.736,Z 365.655,A -85,B 0,C 180,E1 -15285.276,E2 -15285.276} C_VEL
LIN {X 0,Y 319.763,Z 365.652,A -85,B 0,C 180,E1 -15289.873,E2 -15289.873} C_VEL
LIN {X 0,Y 319.94,Z 365.634,A -85,B 0,C 180,E1 -15292.427,E2 -15292.427} C_VEL
LIN {X 0,Y 319.752,Z 365.653,A -85,B 0,C 180,E1 -15294.956,E2 -15294.956} C_VEL
LIN {X 0,Y 319.995,Z 365.621,A -85,B 0,C 180,E1 -15297.483,E2 -15297.483} C_VEL
LIN {X 0,Y 320.157,Z 365.604,A -85,B 0,C 180,E1 -15300,E2 -15300} C_VEL
LIN {X 0,Y 319.995,Z 365.624,A -85,B 0,C 180,E1 -15302.518,E2 -15302.518} C_VEL
LIN {X 0,Y 319.936,Z 365.628,A -85,B 0,C 180,E1 -15306.672,E2 -15306.672} C_VEL
LIN {X 0,Y 319.764,Z 365.655,A -85,B 0,C 180,E1 -15310.127,E2 -15310.127} C_VEL
LIN {X 0,Y 319.737,Z 365.652,A -85,B 0,C 180,E1 -15314.724,E2 -15314.724} C_VEL
LIN {X 0,Y 319.695,Z 365.659,A -85,B 0,C 180,E1 -15319.038,E2 -15319.038} C_VEL
LIN {X 0,Y 319.577,Z 365.674,A -85,B 0,C 180,E1 -15323.319,E2 -15323.319} C_VEL
LIN {X 0,Y 319.64,Z 365.669,A -85,B 0,C 180,E1 -15326.088,E2 -15326.088} C_VEL
LIN {X 0,Y 319.594,Z 365.672,A -85,B 0,C 180,E1 -15328.934,E2 -15328.934} C_VEL
LIN {X 0,Y 319.538,Z 365.682,A -85,B 0,C 180,E1 -15331.862,E2 -15331.862} C_VEL
LIN {X 0,Y 319.587,Z 365.678,A -85,B 0,C 180,E1 -15335.543,E2 -15335.543} C_VEL
LIN {X 0,Y 319.58,Z 365.675,A -85,B 0,C 180,E1 -15338.008,E2 -15338.008} C_VEL
LIN {X 0,Y 319.532,Z 365.683,A -85,B 0,C 180,E1 -15341.597,E2 -15341.597} C_VEL
LIN {X 0,Y 319.521,Z 365.685,A -85,B 0,C 180,E1 -15345.262,E2 -15345.262} C_VEL
LIN {X 0,Y 319.534,Z 365.68,A -85,B 0,C 180,E1 -15348.712,E2 -15348.712} C_VEL
LIN {X 0,Y 319.567,Z 365.675,A -85,B 0,C 180,E1 -15352.348,E2 -15352.348} C_VEL
LIN {X 0,Y 319.566,Z 365.68,A -85,B 0,C 180,E1 -15355.123,E2 -15355.123} C_VEL
LIN {X 0,Y 319.576,Z 365.68,A -85,B 0,C 180,E1 -15359.057,E2 -15359.057} C_VEL
LIN {X 0,Y 319.614,Z 365.671,A -85,B 0,C 180,E1 -15362.498,E2 -15362.498} C_VEL
LIN {X 0,Y 319.611,Z 365.672,A -85,B 0,C 180,E1 -15365.304,E2 -15365.304} C_VEL
LIN {X 0,Y 319.604,Z 365.671,A -85,B 0,C 180,E1 -15368.047,E2 -15368.047} C_VEL
LIN {X 0,Y 319.695,Z 365.665,A -85,B 0,C 180,E1 -15370.962,E2 -15370.962} C_VEL
LIN {X 0,Y 319.737,Z 365.657,A -85,B 0,C 180,E1 -15375.275,E2 -15375.275} C_VEL
LIN {X 0,Y 319.728,Z 365.659,A -85,B 0,C 180,E1 -15377.099,E2 -15377.099} C_VEL
LIN {X 0,Y 324.111,Z 379.417,A -85,B 0,C 180,E1 -15378.302,E2 -15378.302} C_VEL
LIN {X 0,Y 326.503,Z 387.916,A -85,B 0,C 180,E1 -15379.193,E2 -15379.193} C_VEL
LIN {X 0,Y 325.449,Z 399.342,A -85,B 0,C 180,E1 -15380.365,E2 -15380.365} C_VEL
LIN {X 0,Y 324.399,Z 409.89,A -85,B 0,C 180,E1 -15381.747,E2 -15381.747} C_VEL
LIN {X 0,Y 323.347,Z 420.243,A -85,B 0,C 180,E1 -15383.447,E2 -15383.447} C_VEL
LIN {X 0,Y 322.228,Z 429.227,A -85,B 0,C 180,E1 -15385.308,E2 -15385.308} C_VEL
LIN {X 0,Y 321.263,Z 436.473,A -85,B 0,C 180,E1 -15387.178,E2 -15387.178} C_VEL
LIN {X 0,Y 320.446,Z 443.131,A -85,B 0,C 180,E1 -15389.371,E2 -15389.371} C_VEL
LIN {X 0,Y 319.946,Z 447.529,A -85,B 0,C 180,E1 -15391.258,E2 -15391.258} C_VEL
LIN {X 0,Y 319.57,Z 449.875,A -85,B 0,C 180,E1 -15392.52,E2 -15392.52} C_VEL
LIN {X 0,Y 319.38,Z 451.786,A -85,B 0,C 180,E1 -15393.784,E2 -15393.784} C_VEL
LIN {X 0,Y 319.406,Z 453.264,A -85,B 0,C 180,E1 -15395.048,E2 -15395.048} C_VEL
LIN {X 0,Y 319.364,Z 454.318,A -85,B 0,C 180,E1 -15396.316,E2 -15396.316} C_VEL
LIN {X 0,Y 319.331,Z 455.31,A -85,B 0,C 180,E1 -15398.861,E2 -15398.861} C_VEL
LIN {X 0,Y 319.435,Z 455.225,A -85,B 0,C 180,E1 -15400.137,E2 -15400.137} C_VEL
LIN {X 0,Y 319.845,Z 453.812,A -85,B 0,C 180,E1 -15402.692,E2 -15402.692} C_VEL
LIN {X 0,Y 320.222,Z 452.516,A -85,B 0,C 180,E1 -15403.969,E2 -15403.969} C_VEL
LIN {X 0,Y 320.874,Z 449.746,A -85,B 0,C 180,E1 -15405.888,E2 -15405.888} C_VEL
LIN {X 0,Y 321.739,Z 445.93,A -85,B 0,C 180,E1 -15407.806,E2 -15407.806} C_VEL
LIN {X 0,Y 322.776,Z 440.959,A -85,B 0,C 180,E1 -15409.723,E2 -15409.723} C_VEL
LIN {X 0,Y 324.045,Z 434.629,A -85,B 0,C 180,E1 -15411.635,E2 -15411.635} C_VEL
LIN {X 0,Y 325.565,Z 426.655,A -85,B 0,C 180,E1 -15413.537,E2 -15413.537} C_VEL
LIN {X 0,Y 326.968,Z 418.463,A -85,B 0,C 180,E1 -15415.119,E2 -15415.119} C_VEL
LIN {X 0,Y 328.447,Z 408.367,A -85,B 0,C 180,E1 -15416.701,E2 -15416.701} C_VEL
LIN {X 0,Y 329.911,Z 396.98,A -85,B 0,C 180,E1 -15418.099,E2 -15418.099} C_VEL
LIN {X 0,Y 330.026,Z 393.945,A -85,B 0,C 180,E1 -15418.442,E2 -15418.442} C_VEL
LIN {X 0,Y 326.876,Z 383.959,A -85,B 0,C 180,E1 -15419.732,E2 -15419.732} C_VEL
LIN {X 0,Y 322.689,Z 373.43,A -85,B 0,C 180,E1 -15420.956,E2 -15420.956} C_VEL
LIN {X 0,Y 319.612,Z 365.922,A -85,B 0,C 180,E1 -15421.72,E2 -15421.72} C_VEL
LIN {X 0,Y 319.566,Z 365.683,A -85,B 0,C 180,E1 -15421.857,E2 -15421.857} C_VEL
LIN {X 0,Y 319.58,Z 365.682,A -85,B 0,C 180,E1 -15425.542,E2 -15425.542} C_VEL
LIN {X 0,Y 319.557,Z 365.68,A -85,B 0,C 180,E1 -15428.009,E2 -15428.009} C_VEL
LIN {X 0,Y 319.525,Z 365.683,A -85,B 0,C 180,E1 -15431.596,E2 -15431.596} C_VEL
LIN {X 0,Y 319.493,Z 365.69,A -85,B 0,C 180,E1 -15435.257,E2 -15435.257} C_VEL
LIN {X 0,Y 319.567,Z 365.683,A -85,B 0,C 180,E1 -15438.393,E2 -15438.393} C_VEL
LIN {X 0,Y 319.597,Z 365.678,A -85,B 0,C 180,E1 -15442.338,E2 -15442.338} C_VEL
LIN {X 0,Y 319.559,Z 365.681,A -85,B 0,C 180,E1 -15445.123,E2 -15445.123} C_VEL
LIN {X 0,Y 319.572,Z 365.647,A -85,B 0,C 180,E1 -15449.056,E2 -15449.056} C_VEL
LIN {X 0,Y 319.607,Z 365.664,A -85,B 0,C 180,E1 -15452.497,E2 -15452.497} C_VEL
LIN {X 0,Y 319.602,Z 365.672,A -85,B 0,C 180,E1 -15455.303,E2 -15455.303} C_VEL
LIN {X 0,Y 319.601,Z 365.665,A -85,B 0,C 180,E1 -15457.56,E2 -15457.56} C_VEL
LIN {X 0,Y 318.923,Z 365.757,A -85,B 0,C 180,E1 -15458.612,E2 -15458.612} C_VEL
LIN {X 0,Y 316.102,Z 366.109,A -85,B 0,C 180,E1 -15460.326,E2 -15460.326} C_VEL
LIN {X 0,Y 313.717,Z 366.403,A -85,B 0,C 180,E1 -15461.715,E2 -15461.715} C_VEL
LIN {X 0,Y 312.687,Z 366.528,A -85,B 0,C 180,E1 -15462.79,E2 -15462.79} C_VEL
LIN {X 0,Y 312.598,Z 366.539,A -85,B 0,C 180,E1 -15463.154,E2 -15463.154} C_VEL
LIN {X 0,Y 312.691,Z 366.536,A -85,B 0,C 180,E1 -15465.686,E2 -15465.686} C_VEL
LIN {X 0,Y 312.7,Z 366.531,A -85,B 0,C 180,E1 -15469.641,E2 -15469.641} C_VEL
LIN {X 0,Y 312.868,Z 366.512,A -85,B 0,C 180,E1 -15472.254,E2 -15472.254} C_VEL
LIN {X 0,Y 312.716,Z 366.521,A -85,B 0,C 180,E1 -15474.842,E2 -15474.842} C_VEL
LIN {X 0,Y 312.949,Z 366.504,A -85,B 0,C 180,E1 -15477.425,E2 -15477.425} C_VEL
LIN {X 0,Y 313.118,Z 366.471,A -85,B 0,C 180,E1 -15480,E2 -15480} C_VEL
LIN {X 0,Y 312.949,Z 366.504,A -85,B 0,C 180,E1 -15482.574,E2 -15482.574} C_VEL
LIN {X 0,Y 312.906,Z 366.506,A -85,B 0,C 180,E1 -15486.448,E2 -15486.448} C_VEL
LIN {X 0,Y 312.783,Z 366.518,A -85,B 0,C 180,E1 -15489.049,E2 -15489.049} C_VEL
LIN {X 0,Y 312.63,Z 366.54,A -85,B 0,C 180,E1 -15492.991,E2 -15492.991} C_VEL
LIN {X 0,Y 312.634,Z 366.543,A -85,B 0,C 180,E1 -15495.65,E2 -15495.65} C_VEL
LIN {X 0,Y 312.626,Z 366.546,A -85,B 0,C 180,E1 -15499.237,E2 -15499.237} C_VEL
LIN {X 0,Y 312.541,Z 366.556,A -85,B 0,C 180,E1 -15502.79,E2 -15502.79} C_VEL
LIN {X 0,Y 312.599,Z 366.55,A -85,B 0,C 180,E1 -15505.936,E2 -15505.936} C_VEL
LIN {X 0,Y 312.541,Z 366.557,A -85,B 0,C 180,E1 -15509.65,E2 -15509.65} C_VEL
LIN {X 0,Y 312.516,Z 366.559,A -85,B 0,C 180,E1 -15513.689,E2 -15513.689} C_VEL
LIN {X 0,Y 312.55,Z 366.549,A -85,B 0,C 180,E1 -15517.382,E2 -15517.382} C_VEL
LIN {X 0,Y 312.517,Z 366.548,A -85,B 0,C 180,E1 -15519.181,E2 -15519.181} C_VEL
LIN {X 0,Y 313.882,Z 373.066,A -85,B 0,C 180,E1 -15523.071,E2 -15523.071} C_VEL
LIN {X 0,Y 315.199,Z 379.672,A -85,B 0,C 180,E1 -15526.705,E2 -15526.705} C_VEL
LIN {X 0,Y 316.585,Z 387.102,A -85,B 0,C 180,E1 -15530.499,E2 -15530.499} C_VEL
LIN {X 0,Y 316.905,Z 391.145,A -85,B 0,C 180,E1 -15532.409,E2 -15532.409} C_VEL
LIN {X 0,Y 315.166,Z 401.388,A -85,B 0,C 180,E1 -15536.885,E2 -15536.885} C_VEL
LIN {X 0,Y 313.645,Z 412.035,A -85,B 0,C 180,E1 -15541.389,E2 -15541.389} C_VEL
LIN {X 0,Y 312.68,Z 421.001,A -85,B 0,C 180,E1 -15545.11,E2 -15545.11} C_VEL
LIN {X 0,Y 315.613,Z 435.791,A -85,B 0,C 180,E1 -15545.979,E2 -15545.979} C_VEL
LIN {X 0,Y 317.323,Z 448.207,A -85,B 0,C 180,E1 -15546.895,E2 -15546.895} C_VEL
LIN {X 0,Y 318.29,Z 460.812,A -85,B 0,C 180,E1 -15548.03,E2 -15548.03} C_VEL
LIN {X 0,Y 318.402,Z 471.657,A -85,B 0,C 180,E1 -15549.195,E2 -15549.195} C_VEL
LIN {X 0,Y 317.641,Z 482.848,A -85,B 0,C 180,E1 -15550.618,E2 -15550.618} C_VEL
LIN {X 0,Y 315.778,Z 493.067,A -85,B 0,C 180,E1 -15552.181,E2 -15552.181} C_VEL
LIN {X 0,Y 314.308,Z 501.772,A -85,B 0,C 180,E1 -15553.837,E2 -15553.837} C_VEL
LIN {X 0,Y 313.103,Z 509.759,A -85,B 0,C 180,E1 -15555.706,E2 -15555.706} C_VEL
LIN {X 0,Y 312.085,Z 516.473,A -85,B 0,C 180,E1 -15557.648,E2 -15557.648} C_VEL
LIN {X 0,Y 311.454,Z 521.876,A -85,B 0,C 180,E1 -15559.601,E2 -15559.601} C_VEL
LIN {X 0,Y 311.228,Z 526.134,A -85,B 0,C 180,E1 -15561.561,E2 -15561.561} C_VEL
LIN {X 0,Y 311.269,Z 529.349,A -85,B 0,C 180,E1 -15563.519,E2 -15563.519} C_VEL
LIN {X 0,Y 311.353,Z 530.965,A -85,B 0,C 180,E1 -15564.821,E2 -15564.821} C_VEL
LIN {X 0,Y 311.576,Z 532.137,A -85,B 0,C 180,E1 -15566.121,E2 -15566.121} C_VEL
LIN {X 0,Y 311.72,Z 532.895,A -85,B 0,C 180,E1 -15567.416,E2 -15567.416} C_VEL
LIN {X 0,Y 311.73,Z 533.238,A -85,B 0,C 180,E1 -15568.709,E2 -15568.709} C_VEL
LIN {X 0,Y 311.828,Z 533.186,A -85,B 0,C 180,E1 -15570.001,E2 -15570.001} C_VEL
LIN {X 0,Y 311.783,Z 532.665,A -85,B 0,C 180,E1 -15571.293,E2 -15571.293} C_VEL
LIN {X 0,Y 311.785,Z 531.737,A -85,B 0,C 180,E1 -15572.585,E2 -15572.585} C_VEL
LIN {X 0,Y 311.733,Z 530.387,A -85,B 0,C 180,E1 -15573.879,E2 -15573.879} C_VEL
LIN {X 0,Y 311.498,Z 527.477,A -85,B 0,C 180,E1 -15575.828,E2 -15575.828} C_VEL
LIN {X 0,Y 311.397,Z 523.501,A -85,B 0,C 180,E1 -15577.784,E2 -15577.784} C_VEL
LIN {X 0,Y 311.495,Z 517.391,A -85,B 0,C 180,E1 -15580.071,E2 -15580.071} C_VEL
LIN {X 0,Y 311.973,Z 510.677,A -85,B 0,C 180,E1 -15582.028,E2 -15582.028} C_VEL
LIN {X 0,Y 312.767,Z 502.347,A -85,B 0,C 180,E1 -15583.979,E2 -15583.979} C_VEL
LIN {X 0,Y 313.566,Z 494.569,A -85,B 0,C 180,E1 -15585.471,E2 -15585.471} C_VEL
LIN {X 0,Y 314.628,Z 485.701,A -85,B 0,C 180,E1 -15586.882,E2 -15586.882} C_VEL
LIN {X 0,Y 315.531,Z 475.895,A -85,B 0,C 180,E1 -15588.171,E2 -15588.171} C_VEL
LIN {X 0,Y 315.365,Z 465.107,A -85,B 0,C 180,E1 -15589.36,E2 -15589.36} C_VEL
LIN {X 0,Y 314.886,Z 453.634,A -85,B 0,C 180,E1 -15590.38,E2 -15590.38} C_VEL
LIN {X 0,Y 313.919,Z 439.963,A -85,B 0,C 180,E1 -15591.313,E2 -15591.313} C_VEL
LIN {X 0,Y 312.462,Z 426.999,A -85,B 0,C 180,E1 -15591.964,E2 -15591.964} C_VEL
LIN {X 0,Y 311.882,Z 422.449,A -85,B 0,C 180,E1 -15592.177,E2 -15592.177} C_VEL
LIN {X 0,Y 312.618,Z 412.304,A -85,B 0,C 180,E1 -15596.249,E2 -15596.249} C_VEL
LIN {X 0,Y 313.603,Z 402.358,A -85,B 0,C 180,E1 -15600.282,E2 -15600.282} C_VEL
LIN {X 0,Y 314.625,Z 393.391,A -85,B 0,C 180,E1 -15603.949,E2 -15603.949} C_VEL
LIN {X 0,Y 315.663,Z 386.266,A -85,B 0,C 180,E1 -15606.952,E2 -15606.952} C_VEL
LIN {X 0,Y 315.536,Z 382.555,A -85,B 0,C 180,E1 -15608.584,E2 -15608.584} C_VEL
LIN {X 0,Y 314.16,Z 374.918,A -85,B 0,C 180,E1 -15612.155,E2 -15612.155} C_VEL
LIN {X 0,Y 312.558,Z 366.731,A -85,B 0,C 180,E1 -15616.266,E2 -15616.266} C_VEL
LIN {X 0,Y 312.508,Z 366.556,A -85,B 0,C 180,E1 -15619.875,E2 -15619.875} C_VEL
LIN {X 0,Y 312.54,Z 366.553,A -85,B 0,C 180,E1 -15624.051,E2 -15624.051} C_VEL
LIN {X 0,Y 312.508,Z 366.557,A -85,B 0,C 180,E1 -15627.334,E2 -15627.334} C_VEL
LIN {X 0,Y 312.549,Z 366.551,A -85,B 0,C 180,E1 -15631.279,E2 -15631.279} C_VEL
LIN {X 0,Y 312.59,Z 366.55,A -85,B 0,C 180,E1 -15634.711,E2 -15634.711} C_VEL
LIN {X 0,Y 312.592,Z 366.545,A -85,B 0,C 180,E1 -15637.53,E2 -15637.53} C_VEL
LIN {X 0,Y 312.644,Z 366.539,A -85,B 0,C 180,E1 -15641.657,E2 -15641.657} C_VEL
LIN {X 0,Y 312.699,Z 366.532,A -85,B 0,C 180,E1 -15645.687,E2 -15645.687} C_VEL
LIN {X 0,Y 312.707,Z 366.53,A -85,B 0,C 180,E1 -15649.642,E2 -15649.642} C_VEL
LIN {X 0,Y 312.879,Z 366.513,A -85,B 0,C 180,E1 -15652.255,E2 -15652.255} C_VEL
LIN {X 0,Y 312.722,Z 366.529,A -85,B 0,C 180,E1 -15654.843,E2 -15654.843} C_VEL
LIN {X 0,Y 312.996,Z 366.493,A -85,B 0,C 180,E1 -15658.714,E2 -15658.714} C_VEL
LIN {X 0,Y 312.996,Z 366.493,A -85,B 0,C 180,E1 -15661.287,E2 -15661.287} C_VEL
LIN {X 0,Y 312.722,Z 366.527,A -85,B 0,C 180,E1 -15665.158,E2 -15665.158} C_VEL
LIN {X 0,Y 312.878,Z 366.508,A -85,B 0,C 180,E1 -15667.746,E2 -15667.746} C_VEL
LIN {X 0,Y 312.676,Z 366.536,A -85,B 0,C 180,E1 -15671.671,E2 -15671.671} C_VEL
LIN {X 0,Y 312.706,Z 366.527,A -85,B 0,C 180,E1 -15674.888,E2 -15674.888} C_VEL
LIN {X 0,Y 312.637,Z 366.539,A -85,B 0,C 180,E1 -15679.237,E2 -15679.237} C_VEL
LIN {X 0,Y 312.552,Z 366.547,A -85,B 0,C 180,E1 -15682.789,E2 -15682.789} C_VEL
LIN {X 0,Y 312.609,Z 366.546,A -85,B 0,C 180,E1 -15685.935,E2 -15685.935} C_VEL
LIN {X 0,Y 312.551,Z 366.552,A -85,B 0,C 180,E1 -15689.65,E2 -15689.65} C_VEL
LIN {X 0,Y 312.525,Z 366.557,A -85,B 0,C 180,E1 -15693.689,E2 -15693.689} C_VEL
LIN {X 0,Y 312.544,Z 366.555,A -85,B 0,C 180,E1 -15697.383,E2 -15697.383} C_VEL
LIN {X 0,Y 312.496,Z 366.556,A -85,B 0,C 180,E1 -15700.709,E2 -15700.709} C_VEL
LIN {X 0,Y 312.478,Z 366.558,A -85,B 0,C 180,E1 -15704.206,E2 -15704.206} C_VEL
LIN {X 0,Y 312.492,Z 366.557,A -85,B 0,C 180,E1 -15707.918,E2 -15707.918} C_VEL
LIN {X 0,Y 312.511,Z 366.554,A -85,B 0,C 180,E1 -15711.917,E2 -15711.917} C_VEL
LIN {X 0,Y 312.538,Z 366.551,A -85,B 0,C 180,E1 -15714.22,E2 -15714.22} C_VEL
LIN {X 0,Y 312.51,Z 366.558,A -85,B 0,C 180,E1 -15717.333,E2 -15717.333} C_VEL
LIN {X 0,Y 312.558,Z 366.552,A -85,B 0,C 180,E1 -15721.276,E2 -15721.276} C_VEL
LIN {X 0,Y 312.591,Z 366.548,A -85,B 0,C 180,E1 -15724.71,E2 -15724.71} C_VEL
LIN {X 0,Y 312.593,Z 366.545,A -85,B 0,C 180,E1 -15727.528,E2 -15727.528} C_VEL
LIN {X 0,Y 312.644,Z 366.539,A -85,B 0,C 180,E1 -15731.656,E2 -15731.656} C_VEL
LIN {X 0,Y 312.699,Z 366.532,A -85,B 0,C 180,E1 -15735.686,E2 -15735.686} C_VEL
LIN {X 0,Y 312.669,Z 366.538,A -85,B 0,C 180,E1 -15736.679,E2 -15736.679} C_VEL
LIN {X 0,Y 316.865,Z 379.416,A -85,B 0,C 180,E1 -15737.835,E2 -15737.835} C_VEL
LIN {X 0,Y 319.658,Z 389.469,A -85,B 0,C 180,E1 -15738.908,E2 -15738.908} C_VEL
LIN {X 0,Y 318.522,Z 401.115,A -85,B 0,C 180,E1 -15740.153,E2 -15740.153} C_VEL
LIN {X 0,Y 317.501,Z 411.496,A -85,B 0,C 180,E1 -15741.566,E2 -15741.566} C_VEL
LIN {X 0,Y 316.395,Z 421.695,A -85,B 0,C 180,E1 -15743.302,E2 -15743.302} C_VEL
LIN {X 0,Y 315.231,Z 430.57,A -85,B 0,C 180,E1 -15745.203,E2 -15745.203} C_VEL
LIN {X 0,Y 314.245,Z 437.734,A -85,B 0,C 180,E1 -15747.115,E2 -15747.115} C_VEL
LIN {X 0,Y 313.405,Z 444.285,A -85,B 0,C 180,E1 -15749.357,E2 -15749.357} C_VEL
LIN {X 0,Y 312.906,Z 448.617,A -85,B 0,C 180,E1 -15751.286,E2 -15751.286} C_VEL
LIN {X 0,Y 312.508,Z 450.937,A -85,B 0,C 180,E1 -15752.577,E2 -15752.577} C_VEL
LIN {X 0,Y 312.335,Z 452.816,A -85,B 0,C 180,E1 -15753.87,E2 -15753.87} C_VEL
LIN {X 0,Y 312.375,Z 454.236,A -85,B 0,C 180,E1 -15755.162,E2 -15755.162} C_VEL
LIN {X 0,Y 312.275,Z 455.921,A -85,B 0,C 180,E1 -15757.76,E2 -15757.76} C_VEL
LIN {X 0,Y 312.321,Z 456.2,A -85,B 0,C 180,E1 -15759.062,E2 -15759.062} C_VEL
LIN {X 0,Y 312.429,Z 456.061,A -85,B 0,C 180,E1 -15760.366,E2 -15760.366} C_VEL
LIN {X 0,Y 312.879,Z 454.592,A -85,B 0,C 180,E1 -15762.98,E2 -15762.98} C_VEL
LIN {X 0,Y 313.301,Z 453.263,A -85,B 0,C 180,E1 -15764.284,E2 -15764.284} C_VEL
LIN {X 0,Y 314.004,Z 450.436,A -85,B 0,C 180,E1 -15766.246,E2 -15766.246} C_VEL
LIN {X 0,Y 314.914,Z 446.558,A -85,B 0,C 180,E1 -15768.205,E2 -15768.205} C_VEL
LIN {X 0,Y 316.045,Z 441.505,A -85,B 0,C 180,E1 -15770.161,E2 -15770.161} C_VEL
LIN {X 0,Y 317.391,Z 435.076,A -85,B 0,C 180,E1 -15772.112,E2 -15772.112} C_VEL
LIN {X 0,Y 318.99,Z 427.013,A -85,B 0,C 180,E1 -15774.053,E2 -15774.053} C_VEL
LIN {X 0,Y 320.608,Z 417.914,A -85,B 0,C 180,E1 -15775.807,E2 -15775.807} C_VEL
LIN {X 0,Y 322.025,Z 408.416,A -85,B 0,C 180,E1 -15777.277,E2 -15777.277} C_VEL
LIN {X 0,Y 323.523,Z 397.287,A -85,B 0,C 180,E1 -15778.651,E2 -15778.651} C_VEL
LIN {X 0,Y 322.918,Z 393.872,A -85,B 0,C 180,E1 -15779.105,E2 -15779.105} C_VEL
LIN {X 0,Y 319.299,Z 383.041,A -85,B 0,C 180,E1 -15780.535,E2 -15780.535} C_VEL
LIN {X 0,Y 314.358,Z 371.242,A -85,B 0,C 180,E1 -15781.929,E2 -15781.929} C_VEL
LIN {X 0,Y 312.555,Z 366.829,A -85,B 0,C 180,E1 -15782.38,E2 -15782.38} C_VEL
LIN {X 0,Y 312.505,Z 366.566,A -85,B 0,C 180,E1 -15782.412,E2 -15782.412} C_VEL
LIN {X 0,Y 312.536,Z 366.558,A -85,B 0,C 180,E1 -15785.949,E2 -15785.949} C_VEL
LIN {X 0,Y 312.503,Z 366.558,A -85,B 0,C 180,E1 -15790.124,E2 -15790.124} C_VEL
LIN {X 0,Y 312.458,Z 366.564,A -85,B 0,C 180,E1 -15793.964,E2 -15793.964} C_VEL
LIN {X 0,Y 312.526,Z 366.559,A -85,B 0,C 180,E1 -15797.909,E2 -15797.909} C_VEL
LIN {X 0,Y 312.556,Z 366.555,A -85,B 0,C 180,E1 -15801.904,E2 -15801.904} C_VEL
LIN {X 0,Y 312.505,Z 366.56,A -85,B 0,C 180,E1 -15805.789,E2 -15805.789} C_VEL
LIN {X 0,Y 312.526,Z 366.526,A -85,B 0,C 180,E1 -15808.854,E2 -15808.854} C_VEL
LIN {X 0,Y 312.572,Z 366.532,A -85,B 0,C 180,E1 -15811.824,E2 -15811.824} C_VEL
LIN {X 0,Y 312.583,Z 366.548,A -85,B 0,C 180,E1 -15814.71,E2 -15814.71} C_VEL
LIN {X 0,Y 312.583,Z 366.539,A -85,B 0,C 180,E1 -15817.539,E2 -15817.539} C_VEL
LIN {X 0,Y 312.635,Z 366.534,A -85,B 0,C 180,E1 -15821.656,E2 -15821.656} C_VEL
LIN {X 0,Y 312.598,Z 366.539,A -85,B 0,C 180,E1 -15823.154,E2 -15823.154} C_VEL
LIN {X 0,Y 311.917,Z 366.632,A -85,B 0,C 180,E1 -15824.23,E2 -15824.23} C_VEL
LIN {X 0,Y 309.063,Z 366.988,A -85,B 0,C 180,E1 -15825.982,E2 -15825.982} C_VEL
LIN {X 0,Y 306.671,Z 367.284,A -85,B 0,C 180,E1 -15827.402,E2 -15827.402} C_VEL
LIN {X 0,Y 305.672,Z 367.411,A -85,B 0,C 180,E1 -15828.502,E2 -15828.502} C_VEL
LIN {X 0,Y 305.604,Z 367.415,A -85,B 0,C 180,E1 -15828.874,E2 -15828.874} C_VEL
LIN {X 0,Y 305.809,Z 367.393,A -85,B 0,C 180,E1 -15832.074,E2 -15832.074} C_VEL
LIN {X 0,Y 305.687,Z 367.395,A -85,B 0,C 180,E1 -15834.723,E2 -15834.723} C_VEL
LIN {X 0,Y 305.958,Z 367.37,A -85,B 0,C 180,E1 -15838.683,E2 -15838.683} C_VEL
LIN {X 0,Y 305.958,Z 367.37,A -85,B 0,C 180,E1 -15841.316,E2 -15841.316} C_VEL
LIN {X 0,Y 305.686,Z 367.399,A -85,B 0,C 180,E1 -15845.276,E2 -15845.276} C_VEL
LIN {X 0,Y 305.809,Z 367.393,A -85,B 0,C 180,E1 -15847.926,E2 -15847.926} C_VEL
LIN {X 0,Y 305.6,Z 367.419,A -85,B 0,C 180,E1 -15851.945,E2 -15851.945} C_VEL
LIN {X 0,Y 305.633,Z 367.412,A -85,B 0,C 180,E1 -15855.035,E2 -15855.035} C_VEL
LIN {X 0,Y 305.573,Z 367.423,A -85,B 0,C 180,E1 -15859.445,E2 -15859.445} C_VEL
LIN {X 0,Y 305.486,Z 367.433,A -85,B 0,C 180,E1 -15863.042,E2 -15863.042} C_VEL
LIN {X 0,Y 305.544,Z 367.43,A -85,B 0,C 180,E1 -15866.228,E2 -15866.228} C_VEL
LIN {X 0,Y 305.492,Z 367.437,A -85,B 0,C 180,E1 -15869.051,E2 -15869.051} C_VEL
LIN {X 0,Y 305.441,Z 367.44,A -85,B 0,C 180,E1 -15871.952,E2 -15871.952} C_VEL
LIN {X 0,Y 305.459,Z 367.437,A -85,B 0,C 180,E1 -15875.113,E2 -15875.113} C_VEL
LIN {X 0,Y 305.498,Z 367.472,A -85,B 0,C 180,E1 -15878.542,E2 -15878.542} C_VEL
LIN {X 0,Y 306.76,Z 373.544,A -85,B 0,C 180,E1 -15882.28,E2 -15882.28} C_VEL
LIN {X 0,Y 308.046,Z 379.943,A -85,B 0,C 180,E1 -15885.944,E2 -15885.944} C_VEL
LIN {X 0,Y 309.338,Z 386.933,A -85,B 0,C 180,E1 -15889.648,E2 -15889.648} C_VEL
LIN {X 0,Y 309.927,Z 390.461,A -85,B 0,C 180,E1 -15891.422,E2 -15891.422} C_VEL
LIN {X 0,Y 309.845,Z 392.853,A -85,B 0,C 180,E1 -15892.55,E2 -15892.55} C_VEL
LIN {X 0,Y 308.148,Z 402.406,A -85,B 0,C 180,E1 -15896.814,E2 -15896.814} C_VEL
LIN {X 0,Y 306.639,Z 412.585,A -85,B 0,C 180,E1 -15901.23,E2 -15901.23} C_VEL
LIN {X 0,Y 305.773,Z 420.024,A -85,B 0,C 180,E1 -15904.419,E2 -15904.419} C_VEL
LIN {X 0,Y 308.723,Z 434.864,A -85,B 0,C 180,E1 -15905.324,E2 -15905.324} C_VEL
LIN {X 0,Y 310.633,Z 448.297,A -85,B 0,C 180,E1 -15906.367,E2 -15906.367} C_VEL
LIN {X 0,Y 311.548,Z 459.891,A -85,B 0,C 180,E1 -15907.451,E2 -15907.451} C_VEL
LIN {X 0,Y 311.61,Z 472.448,A -85,B 0,C 180,E1 -15908.848,E2 -15908.848} C_VEL
LIN {X 0,Y 310.914,Z 482.454,A -85,B 0,C 180,E1 -15910.181,E2 -15910.181} C_VEL
LIN {X 0,Y 308.997,Z 492.562,A -85,B 0,C 180,E1 -15911.777,E2 -15911.777} C_VEL
LIN {X 0,Y 307.467,Z 500.895,A -85,B 0,C 180,E1 -15913.399,E2 -15913.399} C_VEL
LIN {X 0,Y 306.209,Z 509.132,A -85,B 0,C 180,E1 -15915.377,E2 -15915.377} C_VEL
LIN {X 0,Y 305.08,Z 515.793,A -85,B 0,C 180,E1 -15917.36,E2 -15917.36} C_VEL
LIN {X 0,Y 304.412,Z 521.151,A -85,B 0,C 180,E1 -15919.358,E2 -15919.358} C_VEL
LIN {X 0,Y 304.181,Z 525.377,A -85,B 0,C 180,E1 -15921.364,E2 -15921.364} C_VEL
LIN {X 0,Y 304.206,Z 528.638,A -85,B 0,C 180,E1 -15923.423,E2 -15923.423} C_VEL
LIN {X 0,Y 304.508,Z 531.299,A -85,B 0,C 180,E1 -15926.031,E2 -15926.031} C_VEL
LIN {X 0,Y 304.671,Z 532.045,A -85,B 0,C 180,E1 -15927.357,E2 -15927.357} C_VEL
LIN {X 0,Y 304.679,Z 532.373,A -85,B 0,C 180,E1 -15928.679,E2 -15928.679} C_VEL
LIN {X 0,Y 304.782,Z 532.295,A -85,B 0,C 180,E1 -15930.001,E2 -15930.001} C_VEL
LIN {X 0,Y 304.736,Z 531.751,A -85,B 0,C 180,E1 -15931.322,E2 -15931.322} C_VEL
LIN {X 0,Y 304.739,Z 530.806,A -85,B 0,C 180,E1 -15932.645,E2 -15932.645} C_VEL
LIN {X 0,Y 304.66,Z 529.435,A -85,B 0,C 180,E1 -15933.969,E2 -15933.969} C_VEL
LIN {X 0,Y 304.436,Z 526.489,A -85,B 0,C 180,E1 -15935.964,E2 -15935.964} C_VEL
LIN {X 0,Y 304.329,Z 522.472,A -85,B 0,C 180,E1 -15937.966,E2 -15937.966} C_VEL
LIN {X 0,Y 304.454,Z 516.298,A -85,B 0,C 180,E1 -15940.307,E2 -15940.307} C_VEL
LIN {X 0,Y 304.974,Z 509.536,A -85,B 0,C 180,E1 -15942.309,E2 -15942.309} C_VEL
LIN {X 0,Y 305.823,Z 501.154,A -85,B 0,C 180,E1 -15944.303,E2 -15944.303} C_VEL
LIN {X 0,Y 306.548,Z 494.272,A -85,B 0,C 180,E1 -15945.655,E2 -15945.655} C_VEL
LIN {X 0,Y 307.649,Z 485.461,A -85,B 0,C 180,E1 -15947.106,E2 -15947.106} C_VEL
LIN {X 0,Y 308.54,Z 477.117,A -85,B 0,C 180,E1 -15948.253,E2 -15948.253} C_VEL
LIN {X 0,Y 308.374,Z 465.141,A -85,B 0,C 180,E1 -15949.644,E2 -15949.644} C_VEL
LIN {X 0,Y 307.902,Z 452.916,A -85,B 0,C 180,E1 -15950.772,E2 -15950.772} C_VEL
LIN {X 0,Y 307.013,Z 440.038,A -85,B 0,C 180,E1 -15951.684,E2 -15951.684} C_VEL
LIN {X 0,Y 305.573,Z 427.171,A -85,B 0,C 180,E1 -15952.366,E2 -15952.366} C_VEL
LIN {X 0,Y 304.832,Z 421.645,A -85,B 0,C 180,E1 -15952.608,E2 -15952.608} C_VEL
LIN {X 0,Y 305.641,Z 411.672,A -85,B 0,C 180,E1 -15956.726,E2 -15956.726} C_VEL
LIN {X 0,Y 306.742,Z 401.318,A -85,B 0,C 180,E1 -15961.033,E2 -15961.033} C_VEL
LIN {X 0,Y 307.862,Z 392.415,A -85,B 0,C 180,E1 -15964.801,E2 -15964.801} C_VEL
LIN {X 0,Y 308.655,Z 386.938,A -85,B 0,C 180,E1 -15967.161,E2 -15967.161} C_VEL
LIN {X 0,Y 308.551,Z 383.87,A -85,B 0,C 180,E1 -15968.555,E2 -15968.555} C_VEL
LIN {X 0,Y 307.458,Z 377.63,A -85,B 0,C 180,E1 -15971.522,E2 -15971.522} C_VEL
LIN {X 0,Y 305.959,Z 369.973,A -85,B 0,C 180,E1 -15975.406,E2 -15975.406} C_VEL
LIN {X 0,Y 305.498,Z 367.434,A -85,B 0,C 180,E1 -15976.8,E2 -15976.8} C_VEL
LIN {X 0,Y 305.462,Z 367.433,A -85,B 0,C 180,E1 -15979.893,E2 -15979.893} C_VEL
LIN {X 0,Y 305.485,Z 367.432,A -85,B 0,C 180,E1 -15983.632,E2 -15983.632} C_VEL
LIN {X 0,Y 305.469,Z 367.435,A -85,B 0,C 180,E1 -15986.484,E2 -15986.484} C_VEL
LIN {X 0,Y 305.462,Z 367.433,A -85,B 0,C 180,E1 -15989.591,E2 -15989.591} C_VEL
LIN {X 0,Y 305.519,Z 367.43,A -85,B 0,C 180,E1 -15992.609,E2 -15992.609} C_VEL
LIN {X 0,Y 305.513,Z 367.427,A -85,B 0,C 180,E1 -15995.539,E2 -15995.539} C_VEL
LIN {X 0,Y 305.525,Z 367.426,A -85,B 0,C 180,E1 -15999.816,E2 -15999.816} C_VEL
LIN {X 0,Y 305.58,Z 367.424,A -85,B 0,C 180,E1 -16002.604,E2 -16002.604} C_VEL
LIN {X 0,Y 305.654,Z 367.409,A -85,B 0,C 180,E1 -16005.349,E2 -16005.349} C_VEL
LIN {X 0,Y 305.644,Z 367.41,A -85,B 0,C 180,E1 -16009.4,E2 -16009.4} C_VEL
LIN {X 0,Y 305.82,Z 367.391,A -85,B 0,C 180,E1 -16012.075,E2 -16012.075} C_VEL
LIN {X 0,Y 305.694,Z 367.405,A -85,B 0,C 180,E1 -16014.724,E2 -16014.724} C_VEL
LIN {X 0,Y 305.963,Z 367.369,A -85,B 0,C 180,E1 -16018.684,E2 -16018.684} C_VEL
LIN {X 0,Y 305.963,Z 367.37,A -85,B 0,C 180,E1 -16021.317,E2 -16021.317} C_VEL
LIN {X 0,Y 305.855,Z 367.381,A -85,B 0,C 180,E1 -16026.634,E2 -16026.634} C_VEL
LIN {X 0,Y 305.742,Z 367.397,A -85,B 0,C 180,E1 -16029.26,E2 -16029.26} C_VEL
LIN {X 0,Y 305.595,Z 367.416,A -85,B 0,C 180,E1 -16033.296,E2 -16033.296} C_VEL
LIN {X 0,Y 305.6,Z 367.418,A -85,B 0,C 180,E1 -16036.02,E2 -16036.02} C_VEL
LIN {X 0,Y 305.583,Z 367.419,A -85,B 0,C 180,E1 -16039.445,E2 -16039.445} C_VEL
LIN {X 0,Y 305.497,Z 367.426,A -85,B 0,C 180,E1 -16043.041,E2 -16043.041} C_VEL
LIN {X 0,Y 305.538,Z 367.424,A -85,B 0,C 180,E1 -16046.221,E2 -16046.221} C_VEL
LIN {X 0,Y 305.501,Z 367.428,A -85,B 0,C 180,E1 -16049.05,E2 -16049.05} C_VEL
LIN {X 0,Y 305.45,Z 367.436,A -85,B 0,C 180,E1 -16051.952,E2 -16051.952} C_VEL
LIN {X 0,Y 305.469,Z 367.433,A -85,B 0,C 180,E1 -16055.113,E2 -16055.113} C_VEL
LIN {X 0,Y 305.473,Z 367.43,A -85,B 0,C 180,E1 -16058.533,E2 -16058.533} C_VEL
LIN {X 0,Y 305.465,Z 367.432,A -85,B 0,C 180,E1 -16062.586,E2 -16062.586} C_VEL
LIN {X 0,Y 305.449,Z 367.434,A -85,B 0,C 180,E1 -16066.348,E2 -16066.348} C_VEL
LIN {X 0,Y 305.464,Z 367.432,A -85,B 0,C 180,E1 -16069.892,E2 -16069.892} C_VEL
LIN {X 0,Y 305.487,Z 367.431,A -85,B 0,C 180,E1 -16073.631,E2 -16073.631} C_VEL
LIN {X 0,Y 305.471,Z 367.432,A -85,B 0,C 180,E1 -16076.483,E2 -16076.483} C_VEL
LIN {X 0,Y 305.502,Z 367.432,A -85,B 0,C 180,E1 -16080.949,E2 -16080.949} C_VEL
LIN {X 0,Y 305.577,Z 367.419,A -85,B 0,C 180,E1 -16084.087,E2 -16084.087} C_VEL
LIN {X 0,Y 305.507,Z 367.429,A -85,B 0,C 180,E1 -16088.402,E2 -16088.402} C_VEL
LIN {X 0,Y 305.596,Z 367.419,A -85,B 0,C 180,E1 -16091.217,E2 -16091.217} C_VEL
LIN {X 0,Y 305.655,Z 367.411,A -85,B 0,C 180,E1 -16095.348,E2 -16095.348} C_VEL
LIN {X 0,Y 305.653,Z 367.412,A -85,B 0,C 180,E1 -16096.24,E2 -16096.24} C_VEL
LIN {X 0,Y 309.689,Z 379.78,A -85,B 0,C 180,E1 -16097.38,E2 -16097.38} C_VEL
LIN {X 0,Y 312.588,Z 389.928,A -85,B 0,C 180,E1 -16098.489,E2 -16098.489} C_VEL
LIN {X 0,Y 312.631,Z 393.037,A -85,B 0,C 180,E1 -16098.819,E2 -16098.819} C_VEL
LIN {X 0,Y 311.519,Z 404.137,A -85,B 0,C 180,E1 -16100.094,E2 -16100.094} C_VEL
LIN {X 0,Y 310.492,Z 414.125,A -85,B 0,C 180,E1 -16101.539,E2 -16101.539} C_VEL
LIN {X 0,Y 309.406,Z 423.128,A -85,B 0,C 180,E1 -16103.15,E2 -16103.15} C_VEL
LIN {X 0,Y 308.234,Z 431.905,A -85,B 0,C 180,E1 -16105.094,E2 -16105.094} C_VEL
LIN {X 0,Y 307.228,Z 438.986,A -85,B 0,C 180,E1 -16107.049,E2 -16107.049} C_VEL
LIN {X 0,Y 306.564,Z 443.763,A -85,B 0,C 180,E1 -16108.685,E2 -16108.685} C_VEL
LIN {X 0,Y 305.993,Z 448.407,A -85,B 0,C 180,E1 -16110.657,E2 -16110.657} C_VEL
LIN {X 0,Y 305.447,Z 451.993,A -85,B 0,C 180,E1 -16112.637,E2 -16112.637} C_VEL
LIN {X 0,Y 305.291,Z 453.837,A -85,B 0,C 180,E1 -16113.959,E2 -16113.959} C_VEL
LIN {X 0,Y 305.323,Z 455.207,A -85,B 0,C 180,E1 -16115.282,E2 -16115.282} C_VEL
LIN {X 0,Y 305.262,Z 456.835,A -85,B 0,C 180,E1 -16117.939,E2 -16117.939} C_VEL
LIN {X 0,Y 305.297,Z 457.081,A -85,B 0,C 180,E1 -16119.272,E2 -16119.272} C_VEL
LIN {X 0,Y 305.643,Z 456.326,A -85,B 0,C 180,E1 -16121.943,E2 -16121.943} C_VEL
LIN {X 0,Y 305.923,Z 455.374,A -85,B 0,C 180,E1 -16123.28,E2 -16123.28} C_VEL
LIN {X 0,Y 306.376,Z 453.998,A -85,B 0,C 180,E1 -16124.614,E2 -16124.614} C_VEL
LIN {X 0,Y 307.14,Z 451.117,A -85,B 0,C 180,E1 -16126.619,E2 -16126.619} C_VEL
LIN {X 0,Y 308.104,Z 447.174,A -85,B 0,C 180,E1 -16128.622,E2 -16128.622} C_VEL
LIN {X 0,Y 309.333,Z 442.033,A -85,B 0,C 180,E1 -16130.618,E2 -16130.618} C_VEL
LIN {X 0,Y 310.75,Z 435.523,A -85,B 0,C 180,E1 -16132.61,E2 -16132.61} C_VEL
LIN {X 0,Y 312.463,Z 427.369,A -85,B 0,C 180,E1 -16134.588,E2 -16134.588} C_VEL
LIN {X 0,Y 314.041,Z 418.699,A -85,B 0,C 180,E1 -16136.279,E2 -16136.279} C_VEL
LIN {X 0,Y 315.649,Z 408.465,A -85,B 0,C 180,E1 -16137.876,E2 -16137.876} C_VEL
LIN {X 0,Y 317.004,Z 398.877,A -85,B 0,C 180,E1 -16139.079,E2 -16139.079} C_VEL
LIN {X 0,Y 314.972,Z 391.344,A -85,B 0,C 180,E1 -16140.159,E2 -16140.159} C_VEL
LIN {X 0,Y 311.072,Z 380.859,A -85,B 0,C 180,E1 -16141.553,E2 -16141.553} C_VEL
LIN {X 0,Y 306.33,Z 370.024,A -85,B 0,C 180,E1 -16142.843,E2 -16142.843} C_VEL
LIN {X 0,Y 305.479,Z 367.434,A -85,B 0,C 180,E1 -16143.102,E2 -16143.102} C_VEL
LIN {X 0,Y 305.475,Z 367.438,A -85,B 0,C 180,E1 -16146.738,E2 -16146.738} C_VEL
LIN {X 0,Y 305.454,Z 367.438,A -85,B 0,C 180,E1 -16150.599,E2 -16150.599} C_VEL
LIN {X 0,Y 305.425,Z 367.441,A -85,B 0,C 180,E1 -16153.654,E2 -16153.654} C_VEL
LIN {X 0,Y 305.485,Z 367.432,A -85,B 0,C 180,E1 -16157.407,E2 -16157.407} C_VEL
LIN {X 0,Y 305.517,Z 367.433,A -85,B 0,C 180,E1 -16161.603,E2 -16161.603} C_VEL
LIN {X 0,Y 305.461,Z 367.437,A -85,B 0,C 180,E1 -16164.886,E2 -16164.886} C_VEL
LIN {X 0,Y 305.453,Z 367.413,A -85,B 0,C 180,E1 -16168.353,E2 -16168.353} C_VEL
LIN {X 0,Y 305.518,Z 367.399,A -85,B 0,C 180,E1 -16171.113,E2 -16171.113} C_VEL
LIN {X 0,Y 305.569,Z 367.421,A -85,B 0,C 180,E1 -16174.087,E2 -16174.087} C_VEL
LIN {X 0,Y 305.498,Z 367.428,A -85,B 0,C 180,E1 -16178.402,E2 -16178.402} C_VEL
LIN {X 0,Y 305.587,Z 367.414,A -85,B 0,C 180,E1 -16181.217,E2 -16181.217} C_VEL
LIN {X 0,Y 305.646,Z 367.415,A -85,B 0,C 180,E1 -16185.348,E2 -16185.348} C_VEL
LIN {X 0,Y 305.604,Z 367.415,A -85,B 0,C 180,E1 -16188.874,E2 -16188.874} C_VEL
LIN {X 0,Y 304.996,Z 367.492,A -85,B 0,C 180,E1 -16189.975,E2 -16189.975} C_VEL
LIN {X 0,Y 302.233,Z 367.838,A -85,B 0,C 180,E1 -16191.77,E2 -16191.77} C_VEL
LIN {X 0,Y 299.834,Z 368.129,A -85,B 0,C 180,E1 -16193.225,E2 -16193.225} C_VEL
LIN {X 0,Y 298.757,Z 368.258,A -85,B 0,C 180,E1 -16194.351,E2 -16194.351} C_VEL
LIN {X 0,Y 298.645,Z 368.272,A -85,B 0,C 180,E1 -16194.733,E2 -16194.733} C_VEL
LIN {X 0,Y 298.924,Z 368.246,A -85,B 0,C 180,E1 -16198.652,E2 -16198.652} C_VEL
LIN {X 0,Y 298.924,Z 368.246,A -85,B 0,C 180,E1 -16201.347,E2 -16201.347} C_VEL
LIN {X 0,Y 298.657,Z 368.274,A -85,B 0,C 180,E1 -16205.401,E2 -16205.401} C_VEL
LIN {X 0,Y 298.754,Z 368.272,A -85,B 0,C 180,E1 -16208.114,E2 -16208.114} C_VEL
LIN {X 0,Y 298.549,Z 368.297,A -85,B 0,C 180,E1 -16212.231,E2 -16212.231} C_VEL
LIN {X 0,Y 298.601,Z 368.289,A -85,B 0,C 180,E1 -16215.209,E2 -16215.209} C_VEL
LIN {X 0,Y 298.535,Z 368.301,A -85,B 0,C 180,E1 -16219.243,E2 -16219.243} C_VEL
LIN {X 0,Y 298.453,Z 368.307,A -85,B 0,C 180,E1 -16223.598,E2 -16223.598} C_VEL
LIN {X 0,Y 298.485,Z 368.309,A -85,B 0,C 180,E1 -16226.575,E2 -16226.575} C_VEL
LIN {X 0,Y 298.417,Z 368.316,A -85,B 0,C 180,E1 -16229.641,E2 -16229.641} C_VEL
LIN {X 0,Y 298.392,Z 368.319,A -85,B 0,C 180,E1 -16232.8,E2 -16232.8} C_VEL
LIN {X 0,Y 298.467,Z 368.31,A -85,B 0,C 180,E1 -16236.814,E2 -16236.814} C_VEL
LIN {X 0,Y 298.479,Z 368.488,A -85,B 0,C 180,E1 -16237.923,E2 -16237.923} C_VEL
LIN {X 0,Y 299.791,Z 374.829,A -85,B 0,C 180,E1 -16241.967,E2 -16241.967} C_VEL
LIN {X 0,Y 301.004,Z 380.909,A -85,B 0,C 180,E1 -16245.538,E2 -16245.538} C_VEL
LIN {X 0,Y 302.309,Z 387.98,A -85,B 0,C 180,E1 -16249.389,E2 -16249.389} C_VEL
LIN {X 0,Y 302.941,Z 391.507,A -85,B 0,C 180,E1 -16251.218,E2 -16251.218} C_VEL
LIN {X 0,Y 302.983,Z 393.212,A -85,B 0,C 180,E1 -16252.061,E2 -16252.061} C_VEL
LIN {X 0,Y 301.159,Z 403.256,A -85,B 0,C 180,E1 -16256.67,E2 -16256.67} C_VEL
LIN {X 0,Y 299.559,Z 413.533,A -85,B 0,C 180,E1 -16261.253,E2 -16261.253} C_VEL
LIN {X 0,Y 298.836,Z 419.148,A -85,B 0,C 180,E1 -16263.701,E2 -16263.701} C_VEL
LIN {X 0,Y 301.825,Z 433.544,A -85,B 0,C 180,E1 -16264.613,E2 -16264.613} C_VEL
LIN {X 0,Y 303.546,Z 444.956,A -85,B 0,C 180,E1 -16265.508,E2 -16265.508} C_VEL
LIN {X 0,Y 304.652,Z 457.207,A -85,B 0,C 180,E1 -16266.652,E2 -16266.652} C_VEL
LIN {X 0,Y 304.907,Z 468.612,A -85,B 0,C 180,E1 -16267.92,E2 -16267.92} C_VEL
LIN {X 0,Y 304.354,Z 479.705,A -85,B 0,C 180,E1 -16269.382,E2 -16269.382} C_VEL
LIN {X 0,Y 303.049,Z 488.288,A -85,B 0,C 180,E1 -16270.704,E2 -16270.704} C_VEL
LIN {X 0,Y 301.2,Z 497.205,A -85,B 0,C 180,E1 -16272.343,E2 -16272.343} C_VEL
LIN {X 0,Y 299.766,Z 505.219,A -85,B 0,C 180,E1 -16274.16,E2 -16274.16} C_VEL
LIN {X 0,Y 298.538,Z 511.98,A -85,B 0,C 180,E1 -16276.038,E2 -16276.038} C_VEL
LIN {X 0,Y 297.807,Z 516.994,A -85,B 0,C 180,E1 -16277.738,E2 -16277.738} C_VEL
LIN {X 0,Y 297.259,Z 521.921,A -85,B 0,C 180,E1 -16279.787,E2 -16279.787} C_VEL
LIN {X 0,Y 297.061,Z 525.751,A -85,B 0,C 180,E1 -16281.84,E2 -16281.84} C_VEL
LIN {X 0,Y 297.13,Z 528.041,A -85,B 0,C 180,E1 -16283.425,E2 -16283.425} C_VEL
LIN {X 0,Y 297.441,Z 530.462,A -85,B 0,C 180,E1 -16285.936,E2 -16285.936} C_VEL
LIN {X 0,Y 297.622,Z 531.195,A -85,B 0,C 180,E1 -16287.294,E2 -16287.294} C_VEL
LIN {X 0,Y 297.629,Z 531.507,A -85,B 0,C 180,E1 -16288.648,E2 -16288.648} C_VEL
LIN {X 0,Y 297.737,Z 531.398,A -85,B 0,C 180,E1 -16290.001,E2 -16290.001} C_VEL
LIN {X 0,Y 297.688,Z 530.838,A -85,B 0,C 180,E1 -16291.354,E2 -16291.354} C_VEL
LIN {X 0,Y 297.692,Z 529.876,A -85,B 0,C 180,E1 -16292.707,E2 -16292.707} C_VEL
LIN {X 0,Y 297.589,Z 528.484,A -85,B 0,C 180,E1 -16294.064,E2 -16294.064} C_VEL
LIN {X 0,Y 297.376,Z 525.502,A -85,B 0,C 180,E1 -16296.106,E2 -16296.106} C_VEL
LIN {X 0,Y 297.252,Z 521.44,A -85,B 0,C 180,E1 -16298.156,E2 -16298.156} C_VEL
LIN {X 0,Y 297.407,Z 515.2,A -85,B 0,C 180,E1 -16300.554,E2 -16300.554} C_VEL
LIN {X 0,Y 297.983,Z 508.391,A -85,B 0,C 180,E1 -16302.602,E2 -16302.602} C_VEL
LIN {X 0,Y 298.83,Z 499.942,A -85,B 0,C 180,E1 -16304.646,E2 -16304.646} C_VEL
LIN {X 0,Y 299.737,Z 492.668,A -85,B 0,C 180,E1 -16306.086,E2 -16306.086} C_VEL
LIN {X 0,Y 300.971,Z 483.028,A -85,B 0,C 180,E1 -16307.673,E2 -16307.673} C_VEL
LIN {X 0,Y 301.532,Z 475.628,A -85,B 0,C 180,E1 -16308.693,E2 -16308.693} C_VEL
LIN {X 0,Y 301.413,Z 465.165,A -85,B 0,C 180,E1 -16309.939,E2 -16309.939} C_VEL
LIN {X 0,Y 301,Z 452.672,A -85,B 0,C 180,E1 -16311.14,E2 -16311.14} C_VEL
LIN {X 0,Y 300.086,Z 439.297,A -85,B 0,C 180,E1 -16312.121,E2 -16312.121} C_VEL
LIN {X 0,Y 298.491,Z 425.634,A -85,B 0,C 180,E1 -16312.867,E2 -16312.867} C_VEL
LIN {X 0,Y 297.807,Z 420.772,A -85,B 0,C 180,E1 -16313.092,E2 -16313.092} C_VEL
LIN {X 0,Y 298.678,Z 410.817,A -85,B 0,C 180,E1 -16317.314,E2 -16317.314} C_VEL
LIN {X 0,Y 299.674,Z 402.049,A -85,B 0,C 180,E1 -16321.062,E2 -16321.062} C_VEL
LIN {X 0,Y 300.937,Z 392.595,A -85,B 0,C 180,E1 -16325.177,E2 -16325.177} C_VEL
LIN {X 0,Y 301.655,Z 387.103,A -85,B 0,C 180,E1 -16327.614,E2 -16327.614} C_VEL
LIN {X 0,Y 301.204,Z 382.818,A -85,B 0,C 180,E1 -16329.647,E2 -16329.647} C_VEL
LIN {X 0,Y 299.805,Z 375.309,A -85,B 0,C 180,E1 -16333.39,E2 -16333.39} C_VEL
LIN {X 0,Y 298.447,Z 368.312,A -85,B 0,C 180,E1 -16337.159,E2 -16337.159} C_VEL
LIN {X 0,Y 298.408,Z 368.316,A -85,B 0,C 180,E1 -16341.007,E2 -16341.007} C_VEL
LIN {X 0,Y 298.423,Z 368.312,A -85,B 0,C 180,E1 -16343.931,E2 -16343.931} C_VEL
LIN {X 0,Y 298.398,Z 368.314,A -85,B 0,C 180,E1 -16347.984,E2 -16347.984} C_VEL
LIN {X 0,Y 298.462,Z 368.305,A -85,B 0,C 180,E1 -16351.904,E2 -16351.904} C_VEL
LIN {X 0,Y 298.488,Z 368.306,A -85,B 0,C 180,E1 -16354.924,E2 -16354.924} C_VEL
LIN {X 0,Y 298.456,Z 368.307,A -85,B 0,C 180,E1 -16359.316,E2 -16359.316} C_VEL
LIN {X 0,Y 298.543,Z 368.298,A -85,B 0,C 180,E1 -16362.18,E2 -16362.18} C_VEL
LIN {X 0,Y 298.599,Z 368.29,A -85,B 0,C 180,E1 -16364.995,E2 -16364.995} C_VEL
LIN {X 0,Y 298.599,Z 368.288,A -85,B 0,C 180,E1 -16369.147,E2 -16369.147} C_VEL
LIN {X 0,Y 298.766,Z 368.268,A -85,B 0,C 180,E1 -16371.886,E2 -16371.886} C_VEL
LIN {X 0,Y 298.665,Z 368.282,A -85,B 0,C 180,E1 -16374.599,E2 -16374.599} C_VEL
LIN {X 0,Y 298.929,Z 368.245,A -85,B 0,C 180,E1 -16378.653,E2 -16378.653} C_VEL
LIN {X 0,Y 298.929,Z 368.246,A -85,B 0,C 180,E1 -16381.347,E2 -16381.347} C_VEL
LIN {X 0,Y 298.804,Z 368.258,A -85,B 0,C 180,E1 -16386.754,E2 -16386.754} C_VEL
LIN {X 0,Y 298.687,Z 368.276,A -85,B 0,C 180,E1 -16389.481,E2 -16389.481} C_VEL
LIN {X 0,Y 298.558,Z 368.294,A -85,B 0,C 180,E1 -16393.615,E2 -16393.615} C_VEL
LIN {X 0,Y 298.555,Z 368.293,A -85,B 0,C 180,E1 -16396.409,E2 -16396.409} C_VEL
LIN {X 0,Y 298.518,Z 368.301,A -85,B 0,C 180,E1 -16399.655,E2 -16399.655} C_VEL
LIN {X 0,Y 298.464,Z 368.305,A -85,B 0,C 180,E1 -16403.598,E2 -16403.598} C_VEL
LIN {X 0,Y 298.493,Z 368.301,A -85,B 0,C 180,E1 -16406.575,E2 -16406.575} C_VEL
LIN {X 0,Y 298.426,Z 368.311,A -85,B 0,C 180,E1 -16409.641,E2 -16409.641} C_VEL
LIN {X 0,Y 298.402,Z 368.312,A -85,B 0,C 180,E1 -16412.8,E2 -16412.8} C_VEL
LIN {X 0,Y 298.471,Z 368.304,A -85,B 0,C 180,E1 -16416.812,E2 -16416.812} C_VEL
LIN {X 0,Y 298.394,Z 368.315,A -85,B 0,C 180,E1 -16421.088,E2 -16421.088} C_VEL
LIN {X 0,Y 298.394,Z 368.315,A -85,B 0,C 180,E1 -16425.041,E2 -16425.041} C_VEL
LIN {X 0,Y 298.394,Z 368.315,A -85,B 0,C 180,E1 -16428.912,E2 -16428.912} C_VEL
LIN {X 0,Y 298.452,Z 368.31,A -85,B 0,C 180,E1 -16433.192,E2 -16433.192} C_VEL
LIN {X 0,Y 298.401,Z 368.317,A -85,B 0,C 180,E1 -16437.199,E2 -16437.199} C_VEL
LIN {X 0,Y 298.438,Z 368.31,A -85,B 0,C 180,E1 -16440.614,E2 -16440.614} C_VEL
LIN {X 0,Y 298.49,Z 368.303,A -85,B 0,C 180,E1 -16443.473,E2 -16443.473} C_VEL
LIN {X 0,Y 298.441,Z 368.311,A -85,B 0,C 180,E1 -16446.697,E2 -16446.697} C_VEL
LIN {X 0,Y 298.545,Z 368.298,A -85,B 0,C 180,E1 -16450.756,E2 -16450.756} C_VEL
LIN {X 0,Y 298.599,Z 368.293,A -85,B 0,C 180,E1 -16454.994,E2 -16454.994} C_VEL
LIN {X 0,Y 298.624,Z 368.287,A -85,B 0,C 180,E1 -16455.779,E2 -16455.779} C_VEL
LIN {X 0,Y 302.913,Z 381.325,A -85,B 0,C 180,E1 -16457.025,E2 -16457.025} C_VEL
LIN {X 0,Y 305.907,Z 391.93,A -85,B 0,C 180,E1 -16458.234,E2 -16458.234} C_VEL
LIN {X 0,Y 304.883,Z 403.362,A -85,B 0,C 180,E1 -16459.54,E2 -16459.54} C_VEL
LIN {X 0,Y 303.788,Z 413.653,A -85,B 0,C 180,E1 -16461.015,E2 -16461.015} C_VEL
LIN {X 0,Y 302.689,Z 422.942,A -85,B 0,C 180,E1 -16462.662,E2 -16462.662} C_VEL
LIN {X 0,Y 301.411,Z 431.912,A -85,B 0,C 180,E1 -16464.647,E2 -16464.647} C_VEL
LIN {X 0,Y 300.334,Z 439.147,A -85,B 0,C 180,E1 -16466.645,E2 -16466.645} C_VEL
LIN {X 0,Y 299.53,Z 444.945,A -85,B 0,C 180,E1 -16468.655,E2 -16468.655} C_VEL
LIN {X 0,Y 298.95,Z 449.523,A -85,B 0,C 180,E1 -16470.673,E2 -16470.673} C_VEL
LIN {X 0,Y 298.388,Z 453.05,A -85,B 0,C 180,E1 -16472.699,E2 -16472.699} C_VEL
LIN {X 0,Y 298.244,Z 454.842,A -85,B 0,C 180,E1 -16474.053,E2 -16474.053} C_VEL
LIN {X 0,Y 298.275,Z 456.178,A -85,B 0,C 180,E1 -16475.407,E2 -16475.407} C_VEL
LIN {X 0,Y 298.218,Z 457.755,A -85,B 0,C 180,E1 -16478.128,E2 -16478.128} C_VEL
LIN {X 0,Y 298.28,Z 457.948,A -85,B 0,C 180,E1 -16479.492,E2 -16479.492} C_VEL
LIN {X 0,Y 298.653,Z 457.137,A -85,B 0,C 180,E1 -16482.226,E2 -16482.226} C_VEL
LIN {X 0,Y 298.977,Z 456.156,A -85,B 0,C 180,E1 -16483.595,E2 -16483.595} C_VEL
LIN {X 0,Y 299.933,Z 453.179,A -85,B 0,C 180,E1 -16486.113,E2 -16486.113} C_VEL
LIN {X 0,Y 300.968,Z 449.218,A -85,B 0,C 180,E1 -16488.374,E2 -16488.374} C_VEL
LIN {X 0,Y 302.143,Z 444.435,A -85,B 0,C 180,E1 -16490.419,E2 -16490.419} C_VEL
LIN {X 0,Y 303.53,Z 438.57,A -85,B 0,C 180,E1 -16492.388,E2 -16492.388} C_VEL
LIN {X 0,Y 305.314,Z 430.691,A -85,B 0,C 180,E1 -16494.477,E2 -16494.477} C_VEL
LIN {X 0,Y 307.099,Z 421.773,A -85,B 0,C 180,E1 -16496.345,E2 -16496.345} C_VEL
LIN {X 0,Y 308.74,Z 412.001,A -85,B 0,C 180,E1 -16498.001,E2 -16498.001} C_VEL
LIN {X 0,Y 310.254,Z 402.292,A -85,B 0,C 180,E1 -16499.314,E2 -16499.314} C_VEL
LIN {X 0,Y 310.485,Z 400.545,A -85,B 0,C 180,E1 -16499.518,E2 -16499.518} C_VEL
LIN {X 0,Y 308.052,Z 392.273,A -85,B 0,C 180,E1 -16500.77,E2 -16500.77} C_VEL
LIN {X 0,Y 304.196,Z 381.927,A -85,B 0,C 180,E1 -16502.195,E2 -16502.195} C_VEL
LIN {X 0,Y 299.364,Z 371.053,A -85,B 0,C 180,E1 -16503.549,E2 -16503.549} C_VEL
LIN {X 0,Y 298.427,Z 368.309,A -85,B 0,C 180,E1 -16503.849,E2 -16503.849} C_VEL
LIN {X 0,Y 298.414,Z 368.314,A -85,B 0,C 180,E1 -16507.757,E2 -16507.757} C_VEL
LIN {X 0,Y 298.384,Z 368.319,A -85,B 0,C 180,E1 -16511.26,E2 -16511.26} C_VEL
LIN {X 0,Y 298.353,Z 368.323,A -85,B 0,C 180,E1 -16515.034,E2 -16515.034} C_VEL
LIN {X 0,Y 298.43,Z 368.31,A -85,B 0,C 180,E1 -16516.925,E2 -16516.925} C_VEL
LIN {X 0,Y 298.43,Z 368.313,A -85,B 0,C 180,E1 -16520.998,E2 -16520.998} C_VEL
LIN {X 0,Y 298.432,Z 368.307,A -85,B 0,C 180,E1 -16523.931,E2 -16523.931} C_VEL
LIN {X 0,Y 298.397,Z 368.298,A -85,B 0,C 180,E1 -16527.981,E2 -16527.981} C_VEL
LIN {X 0,Y 298.461,Z 368.289,A -85,B 0,C 180,E1 -16531.904,E2 -16531.904} C_VEL
LIN {X 0,Y 298.483,Z 368.304,A -85,B 0,C 180,E1 -16534.923,E2 -16534.923} C_VEL
LIN {X 0,Y 298.448,Z 368.31,A -85,B 0,C 180,E1 -16539.315,E2 -16539.315} C_VEL
LIN {X 0,Y 298.535,Z 368.287,A -85,B 0,C 180,E1 -16542.179,E2 -16542.179} C_VEL
LIN {X 0,Y 298.59,Z 368.293,A -85,B 0,C 180,E1 -16544.994,E2 -16544.994} C_VEL
LIN {X 0,Y 298.592,Z 368.291,A -85,B 0,C 180,E1 -16549.146,E2 -16549.146} C_VEL
LIN {X 0,Y 298.755,Z 368.271,A -85,B 0,C 180,E1 -16551.885,E2 -16551.885} C_VEL
LIN {X 0,Y 298.645,Z 368.272,A -85,B 0,C 180,E1 -16554.733,E2 -16554.733} C_VEL
LIN {X 0,Y 297.956,Z 368.367,A -85,B 0,C 180,E1 -16555.86,E2 -16555.86} C_VEL
LIN {X 0,Y 295.262,Z 368.706,A -85,B 0,C 180,E1 -16557.703,E2 -16557.703} C_VEL
LIN {X 0,Y 292.231,Z 369.072,A -85,B 0,C 180,E1 -16559.962,E2 -16559.962} C_VEL
LIN {X 0,Y 291.91,Z 369.114,A -85,B 0,C 180,E1 -16560.74,E2 -16560.74} C_VEL
LIN {X 0,Y 291.795,Z 369.139,A -85,B 0,C 180,E1 -16562.761,E2 -16562.761} C_VEL
LIN {X 0,Y 291.743,Z 369.144,A -85,B 0,C 180,E1 -16566.918,E2 -16566.918} C_VEL
LIN {X 0,Y 291.625,Z 369.15,A -85,B 0,C 180,E1 -16569.712,E2 -16569.712} C_VEL
LIN {X 0,Y 291.518,Z 369.165,A -85,B 0,C 180,E1 -16573.95,E2 -16573.95} C_VEL
LIN {X 0,Y 291.483,Z 369.175,A -85,B 0,C 180,E1 -16576.818,E2 -16576.818} C_VEL
LIN {X 0,Y 291.446,Z 369.182,A -85,B 0,C 180,E1 -16579.875,E2 -16579.875} C_VEL
LIN {X 0,Y 291.396,Z 369.187,A -85,B 0,C 180,E1 -16584.205,E2 -16584.205} C_VEL
LIN {X 0,Y 291.419,Z 369.189,A -85,B 0,C 180,E1 -16587.272,E2 -16587.272} C_VEL
LIN {X 0,Y 291.334,Z 369.199,A -85,B 0,C 180,E1 -16590.437,E2 -16590.437} C_VEL
LIN {X 0,Y 291.341,Z 369.196,A -85,B 0,C 180,E1 -16593.699,E2 -16593.699} C_VEL
LIN {X 0,Y 291.43,Z 369.216,A -85,B 0,C 180,E1 -16597.077,E2 -16597.077} C_VEL
